    ConvData[1].TrussInfo := TrussInfo;
    RunTrussInfo          := TRUE;
ELSIF ConvData[1].State = E_Outfeed_Conveyor_State.BUILD_IN_PROGRESS THEN
    //bad truss data, index forward or cancel if it's already cleared
    result := RaiseMessageBox(Header   := 'Old truss data detected',
                              Message1 := 'Conveyor has data from previous truss',
                              Message2 := 'Select Clear if conveyor is clear and ready for current truss',
                              Message3 := 'Select Index to send old truss out down the line',
                              Message4 := 'WARNING make sure conveyor is clear or has correct truss on it',
                              Message5 := 'If Index is pressed robot will place once truss is clear',
                              Btn1     := 'Clear',
                              Btn3     := 'Index');

    IF result = 1 THEN
        ConvData[1].State := E_Outfeed_Conveyor_State.IDLE;
    ELSIF result = 3 THEN
        ConvData[1].State := E_Outfeed_Conveyor_State.INDEX_PREP;
    END_IF

END_IF
END_METHOD

(*! @summary This method contains code which will execute when this PackML module is in the <b>Aborted</b> state*)
METHOD PROTECTED Aborted
ControlPendant.Light.Flash();
LightStack.WhiteLight.Flash();
LightStack.Siren.TurnOff();

IF _OutfeedAutostopOK AND _MainSafetyOK THEN
    ChangeState(E_PMLCommand.ePMLCommand_Clear);
END_IF

AllStopped := FALSE;
END_METHOD

METHOD PROTECTED Execute
VAR_INPUT
END_VAR

VAR_INST
    ErrorPresent : BOOL;
	Manual_R_TRIG : R_TRIG;
END_VAR

VAR CONSTANT
	TestConveyorSpeed : UDINT := 500;
END_VAR
ErrorPresent := FALSE;

AllStopped := TRUE;

FOR i := 1 TO _MaxConveyorCount DO
    AllStopped := AllStopped AND (ConvData[i].State = E_Outfeed_Conveyor_State.IDLE OR ConvData[i].State = E_Outfeed_Conveyor_State.OCCUPIED);
END_FOR

IF EnableManualConveyorControl AND AllStopped THEN
    ManualModeActive := TRUE;
    HMIControl();
ELSE
    ManualModeActive := FALSE;

    FOR i := 2 TO _MaxConveyorCount DO
        ErrorPresent := Convey_Motors[i].Error;

        IF ErrorPresent THEN
            EXIT;
        END_IF
    END_FOR

    IF _OutfeedAutostopOK AND _MainSafetyOK AND ErrorPresent = FALSE THEN
        OutfeedConveyorLogic();
    ELSE
        ChangeState(E_PMLCommand.ePMLCommand_Suspend);
    END_IF

    StartUp := FALSE;
    SUPER^.Execute();
END_IF

Manual_R_TRIG(CLK := ManualModeActive);

IF Manual_R_TRIG.Q THEN
    FOR i := 1 TO _MaxConveyorCount DO
        ConvData[i].ManualControlSelected := FALSE;
    END_FOR
END_IF
END_METHOD

METHOD PROTECTED Held
VAR_INPUT
END_VAR
IF _OutfeedAutostopOK AND _MainSafetyOK THEN
    ChangeState(E_PMLCommand.ePMLCommand_Unhold);
END_IF

FOR i := 1 TO _MaxConveyorCount DO
    ConvData[i].SubState := CONV_MOVE_ASSIGN;
END_FOR
END_METHOD

METHOD PROTECTED Idle
VAR_INPUT
END_VAR
IF _OutfeedAutostopOK AND _MainSafetyOK THEN
    ChangeState(E_PMLCommand.ePMLCommand_Start);
END_IF

FOR i := 1 TO _MaxConveyorCount DO
    ConvData[i].SubState := CONV_MOVE_ASSIGN;
END_FOR

EnableManualConveyorControl := FALSE;
END_METHOD

METHOD PROTECTED Stopped
VAR_INPUT
END_VAR
IF _OutfeedAutostopOK AND _MainSafetyOK THEN
    ChangeState(E_PMLCommand.ePMLCommand_Reset);
END_IF

//skip when warm restart detected
RecoveryDetected := NOT StartUp;
END_METHOD

METHOD PROTECTED Suspended
VAR_INPUT
END_VAR
SuspendTON(IN := TRUE, PT := T#2S);

ControlPendant.Light.Flash();
LightStack.WhiteLight.Flash();
LightStack.Siren.TurnOff();

IF _OutfeedAutostopOK AND _MainSafetyOK AND SuspendTON.Q THEN
    ChangeState(E_PMLCommand.ePMLCommand_Unsuspend);
END_IF

FOR i := 1 TO _MaxConveyorCount DO
    ConvData[i].SubState := CONV_MOVE_ASSIGN;
END_FOR

AllStopped := FALSE;
END_METHOD

//! @summary This method monitors <b>components</b> within this PackML module and initiates fault responses as required
METHOD PROTECTED ComponentMonitor : BOOL
VAR
    AlarmResponses : ARRAY[0..4] OF E_AlarmResponse; //Temporary response array
    i              : UDINT;
END_VAR

//! @description This method is called cyclically by <c>CyclicLogic()</c>
FOR i := 2 TO NumberOfComponents DO
    IF _CurrentState <> E_PMLState.ePMLState_Aborted AND
       _CurrentState <> E_PMLState.ePMLState_Aborting AND
       _CurrentState <> E_PMLState.ePMLState_Clearing AND
       _CurrentState <> E_PMLState.ePMLState_Suspended AND
       _CurrentState <> E_PMLState.ePMLState_Unsuspending AND
       _CurrentState <> E_PMLState.ePMLState_Held AND
       _CurrentState <> E_PMLState.ePMLState_Unholding AND
       _CurrentState <> E_PMLState.ePMLState_Stopped AND
       _CurrentState <> E_PMLState.ePMLState_Stopping THEN
        AlarmResponses := ipComponents[i].ParentResponseDefinitions;

        CASE AlarmResponses[ipComponents[i].CurrentAlarmSeverity] OF
            E_AlarmResponse.Abort_ImmediateError:
                SuspendImmediate();

            E_AlarmResponse.Abort_Immediate:
                SuspendControlled();

            E_AlarmResponse.Stop_Immediate:
                StopImmediate();

            E_AlarmResponse.Stop_Controlled:
                StopControlled();

            E_AlarmResponse.Hold_Immediate:
                HoldImmediate();

            E_AlarmResponse.Hold_Controlled:
                HoldControlled();

            E_AlarmResponse.Suspend_Immediate:
                SuspendImmediate();

            E_AlarmResponse.Suspend_Controlled:
                SuspendControlled();

            E_AlarmResponse.NoResponse:
                ;
        END_CASE
    ELSIF _CurrentState = E_PMLState.ePMLState_Stopped OR _CurrentState = E_PMLState.ePMLState_Stopping THEN
        AlarmResponses := ipComponents[i].ParentResponseDefinitions;

        CASE AlarmResponses[ipComponents[i].CurrentAlarmSeverity] OF
            E_AlarmResponse.Abort_ImmediateError:
                AbortImmediateError(ipComponents[i].Name, FALSE);

            E_AlarmResponse.Abort_Immediate:
                AbortImmediate();

            E_AlarmResponse.NoResponse:
                ;
        END_CASE
    END_IF
END_FOR
END_METHOD

METHOD PROTECTED CreateEvents
VAR_INPUT
END_VAR
F_CreateAllEventsInClass(Alarms     := OutfeedJigAlarms,
                         ClassSize  := SIZEOF(TC_EVENTS.Outfeed_Jig),
                         pInitEvent := ADR(TC_EVENTS.Outfeed_Jig.InitReferenceEvent),
                         Prefix     := _Name);

SUPER^.CreateEvents();
END_METHOD

METHOD HMIControl
VAR_INPUT
END_VAR

VAR
	AllReset : BOOL;
END_VAR
IF ManualReset = FALSE THEN

    FOR i := 1 TO _MaxConveyorCount DO

        IF ManualControlConveyFWD THEN
            IF ConvData[i].ManualControlSelected AND ConvData[i].State = E_Outfeed_Conveyor_State.IDLE THEN
                Convey_Motors[i].MoveVelocity(ManualConveyorSpeed, TRUE);
            ELSE
                IF Convey_Motors[i].Busy THEN
                    Convey_Motors[i].Stop();
                END_IF
            END_IF
        ELSIF ManualControlConveyREV THEN
            IF ConvData[i].ManualControlSelected AND ConvData[i].State = E_Outfeed_Conveyor_State.IDLE THEN
                Convey_Motors[i].MoveVelocity(-ManualConveyorSpeed, TRUE);
            ELSE
                IF Convey_Motors[i].Busy THEN
                    Convey_Motors[i].Stop();
                END_IF
            END_IF
        ELSE

            IF Convey_Motors[i].Busy THEN
                Convey_Motors[i].Stop();
            END_IF
        END_IF

    END_FOR
ELSE
	AllReset := TRUE;
    FOR i := 1 TO _MaxConveyorCount DO
       AllReset := MotorResetAndEnable(Convey_Motors[i]) AND AllReset; 
    END_FOR
	IF AllReset THEN
		ManualReset := FALSE;
	END_IF
END_IF
END_METHOD

METHOD IndexFull : BOOL
VAR_INPUT
END_VAR

VAR_INST
    SubState : USINT := 0;
END_VAR
IndexFull := FALSE;

CASE SubState OF
    0:
        IF ConvData[1].State = E_Outfeed_Conveyor_State.BUILD_IN_PROGRESS THEN
            ConvData[1].State := E_Outfeed_Conveyor_State.INDEX_PREP;
            SubState          := 10;
        END_IF

    10:
        IndexFull := TRUE;
        SubState  := 0;

END_CASE
END_METHOD

METHOD IndexHalf : BOOL
VAR_INPUT
END_VAR

VAR_INST
    SubState : USINT := 0;
END_VAR
IndexHalf := FALSE;

CASE SubState OF
    0:
        IF ConvData[1].State = E_Outfeed_Conveyor_State.BUILD_IN_PROGRESS THEN
            ConvData[1].State := E_Outfeed_Conveyor_State.INDEX_HALF_PREP;
        ELSE
            //waiting for conveyor 1 to be in a good spot
        END_IF

        IF ConvData[1].State = E_Outfeed_Conveyor_State.INDEXING_HALF THEN
            SubState := 10;
        END_IF

    10:
        IF ConvData[1].State = E_Outfeed_Conveyor_State.BUILD_IN_PROGRESS THEN
            IndexHalf := TRUE;
            SubState  := 0;
        END_IF

END_CASE
END_METHOD

//! @summary Basic module initialization logic
METHOD PROTECTED Initialize : BOOL;
VAR
    i                        : UDINT;
    varInfo                  : __SYSTEM.VAR_INFO;
    AllSubUnitsInitialized   : BOOL := TRUE;
    AllComponentsInitialized : BOOL := TRUE;
    emptyTrussInfo           : ST_TrussInfo;

END_VAR

//! @description This method is called by <c>CyclicLogic()</c> as required
CASE DescendantSequenceState OF
    0:
        RegisterComponent(Shift_Motors);
        RegisterComponent(ControlPendant);
        RegisterComponent(LightStack);

        FOR i := 1 TO _MaxConveyorCount DO
            RegisterComponent(Convey_Motors[i]);
            //RegisterComponent(Convey_Sensors[i]);
            ConvData[i].SubState           := E_Outfeed_Conveyor_SubState.CONV_MOVE_ASSIGN;
            ConvData[i].HalfIndexCompleted := FALSE;
            ConvData[i].ReadyForSlideOut   := FALSE;
            ConvData[i].ReadyToIndex       := FALSE;
            ConvData[i].ReadyToIndexHalf   := FALSE;
            ConvData[i].ReadyToOutfeed     := FALSE;
            ConvData[i].ReadyToReceive     := FALSE;
        END_FOR

        LogModeChanges  := FALSE;
        LogStateChanges := FALSE;

        RegisterExternalController(Controller := fbControlSourceHMI);
        fbControlSourceHMI.CyclicLogic();

        //Copy Mode names

        FOR i := 1 TO 3 DO
            ModeNames[i] := F_UnitModeToString(UDINT_TO_DINT(i));
        END_FOR

        DescendantSequenceState := 1;

    1:
        CreateEvents();

        IF SUPER^.Initialize() THEN
            DescendantSequenceState := 2;
        END_IF

    2:
        Initialize := TRUE;

END_CASE
END_METHOD

METHOD PROTECTED Monitoring
VAR_INPUT
END_VAR
///////////////////////////////////////////////////////////////////////////////
// 5. Outfeed autostop dropped
///////////////////////////////////////////////////////////////////////////////
IF (NOT OutfeedJigAlarms[E_Outfeed_Jig.OutfeedSafetyDropped].bRaised) AND NOT _OutfeedAutostopOK THEN
    // Raise alarm if Infeed is taking a long time to get a board
    OutfeedJigAlarms[E_Outfeed_Jig.OutfeedSafetyDropped].Raise(0);
ELSIF OutfeedJigAlarms[E_Outfeed_Jig.OutfeedSafetyDropped].bRaised AND _OutfeedAutostopOK THEN
    // Clear when a board is found
    OutfeedJigAlarms[E_Outfeed_Jig.OutfeedSafetyDropped].Clear(0, 0);
END_IF;

///////////////////////////////////////////////////////////////////////////////
// 5. Outfeed autostop dropped
///////////////////////////////////////////////////////////////////////////////
IF (NOT OutfeedJigAlarms[E_Outfeed_Jig.IndexingBlocked].bRaised) AND IndexingBlockedAlarm THEN
    // Raise alarm if Infeed is taking a long time to get a board
    OutfeedJigAlarms[E_Outfeed_Jig.IndexingBlocked].Raise(0);
ELSIF OutfeedJigAlarms[E_Outfeed_Jig.IndexingBlocked].bRaised AND NOT IndexingBlockedAlarm THEN
    // Clear when a board is found
    OutfeedJigAlarms[E_Outfeed_Jig.IndexingBlocked].Clear(0, 0);
END_IF;

//////////////////////////////////////////////////////////////////////////
// Wrap-up: Evaluate overall severity, then run the extended Monitoring
//////////////////////////////////////////////////////////////////////////
_CurrentAlarmSeverity := TcEventSeverity.Verbose;
_CurrentAlarmSeverity := F_GetMaxSeverityRaised(Alarms := OutfeedJigAlarms, CurrentSeverity := _CurrentAlarmSeverity);

// Finally, run the extended monitoring
// SUPER^.Monitoring();
END_METHOD

METHOD MotorsInit : BOOL
VAR_INPUT
END_VAR
MotorsInit := TRUE;

FOR i := 1 TO _MaxConveyorCount DO
    IF (_MainSafetyOK AND _AutostopOK AND i = 1) OR i > 1 THEN
        MotorsInit := MotorResetAndEnable(Convey_Motors[i]) AND MotorsInit AND Shift_Motors.Reset();
    END_IF
END_FOR
END_METHOD

METHOD NewTrussInfo : BOOL
VAR_INPUT
    ConveyorIndex : USINT;
    NewTrussData  : ST_TrussInfo;
END_VAR

VAR
    i              : USINT;
    EmptyBoardData : ST_PickPlace;
    EmptyTrussInfo : ST_TrussInfo;
END_VAR
FOR i := 1 TO 50 DO
    IF ConvData[1].BoardsPresent[i].ID = '' AND ConvData[1].BoardsPresent[i].Length = 0 THEN
        ConvData[1].BoardsPresent[i] := EmptyBoardData;
    END_IF
END_FOR

ConvData[1].TrussInfo := NewTrussData;
END_METHOD

METHOD OutfeedConveyorLogic : BOOL
VAR_INPUT
END_VAR

VAR
    EmptyBoardsPresent : ARRAY[1..50] OF ST_PickPlace;
    EmptyTrussInfo     : ST_TrussInfo;
    TempString         : STRING;
END_VAR

VAR_INST
    Previous_SubState : ARRAY[1..7] OF E_Outfeed_Conveyor_SubState;
    ClearConveyorTON  : TON;
    Previous_State    : ARRAY[1..7] OF E_Outfeed_Conveyor_State;
    Alarm_TON         : ARRAY[1..7] OF TON;
END_VAR
LightStack.WhiteLight.TurnOn();
ControlPendant.Light.TurnOff();

FOR i := 1 TO _MaxConveyorCount DO
    CASE ConvData[i].State OF
        E_Outfeed_Conveyor_State.IDLE:
            ConvData[i].SubState := CONV_MOVE_ASSIGN;

            // check to see if index is requested
            Alarm_TON[i](IN := FALSE, PT := T#5S);

            IF i = _MaxConveyorCount THEN
                ClearConveyorTON(IN := FALSE, PT := T#1000MS);
                LightStack.Siren.TurnOff();
                LightStack.AmberLight.TurnOff();
            END_IF

            IF i > 1 THEN
                IF ConvData[i - 1].ReadyToIndex THEN
                    ConvData[i].State := E_Outfeed_Conveyor_State.RECEIVE_PREP;
                END_IF
            END_IF

        E_Outfeed_Conveyor_State.RECEIVE_PREP:
            // assign absolute position based off relative distance, also sync up with indexing conveyor

            IF Convey_Motors[i].Enabled AND Convey_Motors[i].Error = FALSE THEN
                ConvData[i].TargetPos          := Convey_Motors[i].ActualPosition + ConvData[i].ConveyorLength;
                ConvData[i - 1].ReadyToReceive := TRUE;

                IF i = _MaxConveyorCount AND Shift_Motors.Retracted THEN
                    ConvData[i].State := E_Outfeed_Conveyor_State.RECEIVING;
                ELSE
                    ConvData[i].State := E_Outfeed_Conveyor_State.RECEIVING;
                END_IF
            ELSE
                MotorResetAndEnable(Convey_Motors[i]);
            END_IF

        E_Outfeed_Conveyor_State.RECEIVING:

            // execute movement to position go to RESET when done

            CASE ConvData[i].SubState OF
                CONV_MOVE_ASSIGN:
                    IF i = 2 THEN
                        IF _AutostopOK AND Convey_Motors[i - 1].Axis.Status.DiscreteMotion THEN
                            Convey_Motors[i].MoveAbsolute(ConvData[i].TargetPos, TRUE);
                            ConvData[i].SubState := CONV_MOVE_DONE_CHECK;
                        END_IF
                    ELSE
                        Convey_Motors[i].MoveAbsolute(ConvData[i].TargetPos, TRUE);
                        ConvData[i].SubState := CONV_MOVE_DONE_CHECK;
                    END_IF

                CONV_MOVE_DONE_CHECK:
                    IF Convey_Motors[i].InPosition AND NOT Convey_Motors[i].Busy THEN
                        ConvData[i].SubState := CONV_DATA_CONFIRMATION;
                    ELSIF Convey_Motors[i].Error OR (i = 2 AND (_AutostopOK = FALSE)) THEN
                        ConvData[i].SubState := CONV_RESET_MOTOR;
                    END_IF

                CONV_DATA_CONFIRMATION:
                    Alarm_TON[i](IN := TRUE, PT := T#5S);

                    IF ConvData[i].TrussInfo.TrussID <> '' THEN
                        ConvData[i].SubState := CONV_MOVE_ASSIGN;
                        ConvData[i].State    := E_Outfeed_Conveyor_State.OCCUPIED;
                        Alarm_TON[i](IN := FALSE, PT := T#5S);
                    END_IF

                    Convey_Motors[i].AlarmRaiseBasic(alarm := E_OutfeedConveyor.NoTrussData, raise := Alarm_TON[i].Q);

                CONV_RESET_MOTOR:
                    IF MotorResetAndEnable(Convey_Motors[i]) THEN
                        ConvData[i].SubState := CONV_MOVE_ASSIGN;
                    END_IF
            END_CASE

        E_Outfeed_Conveyor_State.OCCUPIED:
            // check to see if boards can be moved forward

            IF i < _MaxConveyorCount THEN
                IF ConvData[i + 1].State = E_Outfeed_Conveyor_State.IDLE THEN
                    ConvData[i].State := E_Outfeed_Conveyor_State.INDEX_PREP;
                END_IF
            ELSE
                //turn on lights and permissions for extending and retracting conveyor out over table button pressed to clear data and let them retract

                ControlPendant.Light.TurnOn();
                LightStack.AmberLight.TurnOn();
                Shift_Motors.Jog(JogFW := ControlPendant.ExtendSlideout.Button_Pressed, JogBW := ControlPendant.RetractSlideout.Button_Pressed);

                IF Shift_Motors.Retracted = FALSE THEN
                    ConvData[i].State := E_Outfeed_Conveyor_State.RESET;
                ELSIF _InSimulation THEN
                    ConvData[i].State := E_Outfeed_Conveyor_State.AUTO_RETRACT;
                END_IF
            END_IF

        E_Outfeed_Conveyor_State.INDEX_HALF_PREP:
            ConvData[i].TargetPos := Convey_Motors[i].ActualPosition + (ConvData[i].ConveyorLength / 2);
            Alarm_TON[i](IN := TRUE, PT := T#5S);

            // assign absolute position based off relative distance, also sync up with receiving conveyor
            IF Convey_Motors[i].Enabled AND Convey_Motors[i].Error = FALSE THEN
                ConvData[i].State := E_Outfeed_Conveyor_State.INDEXING_HALF;
                Alarm_TON[i](IN := FALSE, PT := T#5S);
            ELSE
                IF _MainSafetyOK AND ((i > 1 AND _OutfeedAutostopOK) OR (i = 1 AND _AutostopOK)) THEN
                    MotorResetAndEnable(Convey_Motors[i]);
                END_IF
            END_IF

            IndexingBlockedAlarm := Alarm_TON[i].Q;

        E_Outfeed_Conveyor_State.INDEXING_HALF:
            // execute movement to position go to RESET when done

            CASE ConvData[i].SubState OF
                CONV_MOVE_ASSIGN:
                    Convey_Motors[i].MoveAbsolute(ConvData[i].TargetPos, TRUE);
                    ConvData[i].SubState := CONV_MOVE_DONE_CHECK;

                CONV_MOVE_DONE_CHECK:
                    IF Convey_Motors[i].InPosition AND NOT Convey_Motors[i].Busy THEN
                        ConvData[i].State    := E_Outfeed_Conveyor_State.BUILD_IN_PROGRESS;
                        ConvData[i].SubState := CONV_MOVE_ASSIGN;
                    ELSIF Convey_Motors[i].Error THEN
                        ConvData[i].SubState := CONV_RESET_MOTOR;
                    END_IF

                CONV_RESET_MOTOR:
                    IF MotorResetAndEnable(Convey_Motors[i]) THEN
                        ConvData[i].SubState := CONV_MOVE_ASSIGN;
                    END_IF

            END_CASE

        E_Outfeed_Conveyor_State.INDEX_PREP:
            Alarm_TON[i](IN := TRUE, PT := T#5S);

            IndexingBlockedAlarm := Alarm_TON[i].Q;

            IF Convey_Motors[i].Enabled AND Convey_Motors[i].Error = FALSE THEN
                ConvData[i].TargetPos    := Convey_Motors[i].ActualPosition + ConvData[i].ConveyorLength;
                ConvData[i].ReadyToIndex := TRUE;

                // assign absolute position based off relative distance, also sync up with receiving conveyor
                IF ConvData[i + 1].State = E_Outfeed_Conveyor_State.RECEIVING THEN
                    IF Convey_Motors[i].Enabled AND Convey_Motors[i].Error = FALSE THEN
                        ConvData[i].State := E_Outfeed_Conveyor_State.INDEXING;
                        Alarm_TON[i](IN := FALSE, PT := T#5S);
                    ELSE
                        MotorResetAndEnable(Convey_Motors[i]);
                    END_IF
                END_IF
            ELSE
                IF _MainSafetyOK AND ((i > 1 AND _OutfeedAutostopOK) OR (i = 1 AND _AutostopOK)) THEN
                    MotorResetAndEnable(Convey_Motors[i]);
                END_IF
            END_IF

        E_Outfeed_Conveyor_State.INDEXING:
            // execute movement to position go to RESET when done

            CASE ConvData[i].SubState OF
                CONV_MOVE_ASSIGN:
                    IF i = 1 THEN
                        IF _AutostopOK THEN
                            Convey_Motors[i].MoveAbsolute(ConvData[i].TargetPos, TRUE);
                            ConvData[i].SubState := CONV_MOVE_DONE_CHECK;
                        END_IF
                    ELSE
                        Convey_Motors[i].MoveAbsolute(ConvData[i].TargetPos, TRUE);
                        ConvData[i].SubState := CONV_MOVE_DONE_CHECK;
                    END_IF

                CONV_MOVE_DONE_CHECK:
                    IF Convey_Motors[i].InPosition AND NOT Convey_Motors[i].Busy THEN
                        ConvData[i].SubState := CONV_DATA_CONFIRMATION;
                    ELSIF Convey_Motors[i].Error OR (i = 1 AND _AutostopOK = FALSE) THEN
                        ConvData[i].SubState := CONV_RESET_MOTOR;
                    END_IF

                CONV_DATA_CONFIRMATION:
                    ConvData[i + 1].BoardsPresent := ConvData[i].BoardsPresent;
                    ConvData[i + 1].TrussInfo     := ConvData[i].TrussInfo;

                    IF ConvData[i + 1].State = E_Outfeed_Conveyor_State.OCCUPIED THEN
                        ConvData[i].State    := E_Outfeed_Conveyor_State.RESET;
                        ConvData[i].SubState := CONV_MOVE_ASSIGN;

                        ConvData[i].ReadyToIndex := FALSE;
                    END_IF

                CONV_RESET_MOTOR:
                    IF MotorResetAndEnable(Convey_Motors[i]) THEN
                        ConvData[i].SubState := CONV_MOVE_ASSIGN;
                    END_IF
            END_CASE

        E_Outfeed_Conveyor_State.RESET:
            // reset data and start at IDLE
            ConvData[i].SubState := CONV_MOVE_ASSIGN;

            IF i < _MaxConveyorCount THEN
                IF Convey_Motors[i].SimHoming(Motor := Convey_Motors[i], SimPos := 0) THEN
                    ConvData[i].BoardsPresent := EmptyBoardsPresent;
                    ConvData[i].TrussInfo     := EmptyTrussInfo;
                    ConvData[i].ReadyToIndex  := FALSE;

                    ConvData[i].State := E_Outfeed_Conveyor_State.IDLE;
                END_IF
            ELSE
                //turn on lights and permissions for extending conveyor out over table, clear data and let them retract

                ClearConveyorTON(IN := ControlPendant.ClearConveyor.Button_Pressed AND ControlPendant.RetractSlideout.Button_Pressed, PT := T#250MS);

                ControlPendant.Light.TurnOn();
                LightStack.AmberLight.TurnOn();
                Shift_Motors.Jog(JogFW := ControlPendant.ExtendSlideout.Button_Pressed, JogBW := ControlPendant.RetractSlideout.Button_Pressed);

                IF ClearConveyorTON.Q THEN
                    ConvData[i].State := E_Outfeed_Conveyor_State.AUTO_RETRACT;
                END_IF

            END_IF

        E_Outfeed_Conveyor_State.AUTO_RETRACT:
            LightStack.AmberLight.Flash();
            LightStack.Siren.Flash();

            IF Shift_Motors.Retracted = FALSE AND _InSimulation = FALSE THEN
                Shift_Motors.Jog(JogFW := FALSE, JogBW := TRUE);

                IF ControlPendant.ExtendSlideout.Button_Pressed THEN
                    ConvData[i].State := E_Outfeed_Conveyor_State.RESET;
                END_IF
            ELSE
                Shift_Motors.Jog(JogFW := FALSE, JogBW := FALSE);

                IF Convey_Motors[i].SimHoming(Motor := Convey_Motors[i], SimPos := 0) THEN
                    ConvData[i].BoardsPresent := EmptyBoardsPresent;
                    ConvData[i].TrussInfo     := EmptyTrussInfo;
                    ConvData[i].ReadyToIndex  := FALSE;
                    ConvData[i].State         := E_Outfeed_Conveyor_State.IDLE;
                    ControlPendant.Light.TurnOff();
                END_IF
            END_IF

        E_Outfeed_Conveyor_State.ERROR:

        // Conveyor errored out, prevent indexing or receiving from other conveyors
    END_CASE

    IF ConvData[i].State <> Previous_State[i] THEN
        TempString := '';
        TempString := CONCAT(TempString, 'Conveyor ');
        TempString := CONCAT(TempString, UDINT_TO_STRING(i));
        TempString := CONCAT(TempString, ' State change to: ');
        Trace(CONCAT(TempString, TO_STRING(ConvData[i].State)));
    END_IF

    Previous_State[i] := ConvData[i].State;

    IF ConvData[i].SubState <> Previous_SubState[i] THEN
        TempString := '';
        TempString := CONCAT(TempString, 'Conveyor ');
        TempString := CONCAT(TempString, UDINT_TO_STRING(i));
        TempString := CONCAT(TempString, ' SubState change to: ');
        Trace(CONCAT(TempString, TO_STRING(ConvData[i].SubState)));
    END_IF

    Previous_SubState[i] := ConvData[i].SubState;

END_FOR
END_METHOD

METHOD PopulateBoardToArray : BOOL
VAR_INPUT
    ConveyorIndex : USINT;
    NewBoardData  : ST_PickPlace;
END_VAR

VAR
    i : USINT;
END_VAR
FOR i := 1 TO 50 DO
    IF ConvData[1].BoardsPresent[i].ID = '' AND ConvData[1].BoardsPresent[i].Length = 0 THEN
        ConvData[1].BoardsPresent[i] := NewBoardData;
        EXIT;
    END_IF
END_FOR
END_METHOD

PROPERTY AutostopOK : bool
SET
_AutostopOK := AutostopOK;
END_SET
END_PROPERTY

PROPERTY MainSafetyOK : bool
SET
_MainSafetyOK := MainSafetyOK;
END_SET
END_PROPERTY

PROPERTY MaxConveyorCount : USINT
SET
_MaxConveyorCount := MaxConveyorCount;
END_SET
END_PROPERTY

PROPERTY OutfeedAutostopOK : bool
SET
_OutfeedAutostopOK := OutfeedAutostopOK;
END_SET
END_PROPERTY

PROPERTY OutfeedConveyorStatus : ST_OutfeedConveyorStatus
GET
OutfeedConveyorStatus := _OutfeedConveyorStatus;
END_GET
END_PROPERTY

PROPERTY ParentState : E_PMLState
SET
_ParentState := ParentState;
END_SET
END_PROPERTY

PROPERTY PickPlace_Done_ENUM : E_WaitSync
SET
_PickPlace_Done_ENUM := PickPlace_Done_ENUM;
END_SET
END_PROPERTY

PROPERTY PickPlace_Ready_ENUM : E_WaitSync
SET
_PickPlace_Ready_ENUM := PickPlace_Ready_ENUM;
END_SET
END_PROPERTY

END_FUNCTION_BLOCK

// Machine/EquipmentModules/Functional Layer/FB_Preplate
FUNCTION_BLOCK FB_Preplate EXTENDS FB_EquipmentModule_SR
VAR
    // Sub module definitions here

    // List of sub modules

    // Component definitions here
    Racks       : ARRAY[1..NUM_OF_PREPLATE_RACKS] OF FB_Component_Preplate_Rack;
    ManDoorLock : FB_Component_Indicator;

END_VAR

VAR CONSTANT

    // Report parameters 

    //Alarms
    NUM_OF_PREPLATE_RACKS : UDINT := 5;

    PREPLATE_ALARM_COUNT : INT := 6;
END_VAR

VAR CONSTANT

    SS_OPEN_DOORS  : INT := 200;
    SS_CLOSE_DOORS : INT := 201;
END_VAR

METHOD CyclicLogic
VAR_INPUT
END_VAR

VAR
    LowLimit  : STRING;
    HighLimit : STRING;
END_VAR
IF NOT _InitComplete THEN
    _InitComplete := Initialize();
    RETURN;
END_IF

SUPER^.CyclicLogic();

IF _CurrentState = E_PMLState.ePMLState_Execute OR
   _CurrentState = E_PMLState.ePMLState_Unholding OR
   _CurrentState = E_PMLState.ePMLState_Unsuspending THEN

    ManDoorLock.TurnOn();
ELSE
    ManDoorLock.TurnOff();
END_IF

IF _CurrentState <> E_PMLState.ePMLState_Execute THEN
    FOR i := 1 TO NUM_OF_PREPLATE_RACKS DO
        Racks[i].Executing := FALSE;
    END_FOR
END_IF

Racks[1].LinkBlocked := Racks[2].Blocked;
Racks[2].LinkBlocked := Racks[1].Blocked;
Racks[3].LinkBlocked := Racks[4].Blocked;
Racks[4].LinkBlocked := Racks[3].Blocked OR Racks[4].Blocked;
Racks[5].LinkBlocked := Racks[4].Blocked;
;
IF NOT Racks[1].IsAvailable() THEN
	Racks[2].Disable();
END_IF

IF NOT Racks[2].IsAvailable() THEN
	Racks[1].Disable();
END_IF

IF NOT Racks[3].IsAvailable() THEN
	Racks[4].Disable();
END_IF

IF NOT Racks[4].IsAvailable() THEN
	Racks[3].Disable();
END_IF

CyclicLogicSimulation();
END_METHOD

(*! @summary This method contains code which will execute when this PackML module is in the <b>Execute</b> state*)
METHOD PROTECTED Execute
ManDoorLock.TurnOn();

FOR i := 1 TO NUM_OF_PREPLATE_RACKS DO
    Racks[i].Executing := TRUE;
END_FOR
END_METHOD

METHOD HMIControl
VAR_INPUT
END_VAR
END_METHOD

//! @summary Basic module initialization logic
METHOD PROTECTED Initialize : BOOL;
VAR
    i                        : UDINT;
    varInfo                  : __SYSTEM.VAR_INFO;
    AllSubUnitsInitialized   : BOOL := TRUE;
    AllComponentsInitialized : BOOL := TRUE;
END_VAR

//! @description This method is called by <c>CyclicLogic()</c> as required
Initialize := FALSE;

CASE DescendantSequenceState OF
    0:
        FOR i := 1 TO NUM_OF_PREPLATE_RACKS DO
            RegisterComponent(Racks[i]);
        END_FOR

        _LogModeChanges         := FALSE;
        _LogStateChanges        := FALSE;
        DescendantSequenceState := DescendantSequenceState + 10;

    10:
        //Setup Custom modes here

        (*CustomModes(eMode                          :=,
                    sName                          :=,
                    bDisableClearing               :=,
                    bDisableStarting               :=,
                    bDisableSuspended              :=,
                    bDisableStopping               :=,
                    bDisableAborting               :=,
                    bDisableHolding                :=,
                    bDisableHeld                   :=,
                    bDisableUnholding              :=,
                    bDisableSuspending             :=,
                    bDisableUnsuspending           :=,
                    bDisableResetting              :=,
                    bDisableIdle                   :=,
                    bDisableCompleting             :=,
                    bDisableComplete               :=,
                    bEnableUnitModeChangeStopped   :=,
                    bEnableUnitModeChangeIdle      :=,
                    bEnableUnitModeChangeSuspended :=,
                    bEnableUnitModeChangeExecute   :=,
                    bEnableUnitModeChangeAborted   :=,
                    bEnableUnitModeChangeHeld      :=,
                    bEnableUnitModeChangeComplete  :=,
                    bError                         =>,
                    nErrorId                       =>);*)

        DescendantSequenceState := DescendantSequenceState + 10;

    20:
        //Copy Mode names

        FOR i := 1 TO 3 DO
            ModeNames[i] := F_UnitModeToString(UDINT_TO_DINT(i));
        END_FOR

        RegisterExternalController(Controller := fbControlSourceHMI);
        fbControlSourceHMI.CyclicLogic();
        DescendantSequenceState := DescendantSequenceState + 10;

    30:
        //Call the Super

        IF SUPER^.Initialize() THEN
            DescendantSequenceState := DescendantSequenceState + 10;
        END_IF

    40:
        Initialize := TRUE;
END_CASE
END_METHOD

PROPERTY PUBLIC InAuto : BOOL
GET
END_GET
SET
FOR i := 1 TO NUM_OF_PREPLATE_RACKS DO
    Racks[i].InAuto := InAuto;
END_FOR
END_SET
END_PROPERTY

END_FUNCTION_BLOCK

// Machine/EquipmentModules/Functional Layer/FB_Press
FUNCTION_BLOCK FB_Press EXTENDS FB_EquipmentModule_SR
VAR
    // Sub module definitions here

    // List of sub modules

    ipSubModules_Init : ARRAY[1..Parameters_PackML_Base.MAX_NO_OF_SUBMODULES] OF I_PackML_BaseModule := [];

    // Component definitions here

    Top_Press    : FB_Component_BasicSlaveAxis_SoE := (Name := 'Top Press');
    Bottom_Press : FB_Component_BasicSlaveAxis_SoE := (Name := 'Bottom Press');

    Top_PressCmds_Extra    : ST_MotorControls_NonStandard;
    Bottom_PressCmds_Extra : ST_MotorControls_NonStandard;

    //Data for recipe

    TopPressRecipe    : ST_PressRecipe;
    BottomPressRecipe : ST_PressRecipe;
    Plates            : ST_Plates;
    DetailIndex       : UDINT := 1;
    Detail_Step       : E_Press_States;

    _NailplateCountData_Ready : BOOL;
    _NailplateCountData_Sent  : BOOL;
    _DriveMode                : SPT_Motion_Control.E_DriveOperationMode;
    _DoublePickDataToPass     : BOOL;
    _DoublePickData_Ready     : BOOL;
    _DoublePickData_Sent      : BOOL;
    _BoardDataToPass          : ST_BoardInfo;
END_VAR

VAR CONSTANT

    // Report parameters 

    FAULTID  : INT := 1; //Fault number 
    CURRTEMP : INT := 2; // current temperature of the sealing bar 
    CURRPOS  : INT := 3; // current position of the sealing bar  

    //Alarms

    PREPLATE_ALARM_COUNT : INT := 6;
END_VAR

VAR
    FB_Reset_SoE_Drive : FB_SoEReset;

    //Robot Signals

    RobotClearOfPress AT %I* : BOOL := TRUE;

    _NailplateDataToPass : ST_PlateInfo;

    TopPressDriveOpMode_Read    : SPT_Motion_Control.MC_ReadDriveOperationMode;
    TopPressDriveOpMode_Write   : SPT_Motion_Control.MC_WriteDriveOperationMode;
    TopPressDriveOpMode_Options : SPT_Motion_Control.ST_DriveOperationModeOptions;

    BottomPressDriveOpMode_Read    : SPT_Motion_Control.MC_ReadDriveOperationMode;
    BottomPressDriveOpMode_Write   : SPT_Motion_Control.MC_WriteDriveOperationMode;
    BottomPressDriveOpMode_Options : SPT_Motion_Control.ST_DriveOperationModeOptions;

    _PressRobotPermissionToEnter : ST_MediatorInterface;
END_VAR

METHOD CyclicLogic
VAR_INPUT
END_VAR

VAR
    LowLimit  : STRING;
    HighLimit : STRING;
END_VAR
IF NOT _InitComplete THEN
    _InitComplete := Initialize();
    RETURN;
END_IF

AllowHMIControl(ThisModuleOnly:=FALSE);

SUPER^.CyclicLogic();
CyclicLogicSimulation();

BottomPressRecipe.AtTop := Bottom_Press.ActualPosition < BottomPressRecipe.OpenPosition + 10;
TopPressRecipe.AtTop    := Top_Press.ActualPosition < TopPressRecipe.OpenPosition + 10;

BottomPressRecipe.AtWork := Bottom_Press.ActualPosition > BottomPressRecipe.ClosedPosition - 10;
TopPressRecipe.AtWork    := Top_Press.ActualPosition > TopPressRecipe.ClosedPosition - 10;

BottomPressRecipe.State_Str := TO_STRING(BottomPressRecipe.State);
BottomPressRecipe.State_Previous_Str := TO_STRING(BottomPressRecipe.State_Previous);
BottomPressRecipe.State_Response_Str := TO_STRING(BottomPressRecipe.State_Response);

TopPressRecipe.State_Str := TO_STRING(TopPressRecipe.State);
TopPressRecipe.State_Previous_Str := TO_STRING(TopPressRecipe.State_Previous);
TopPressRecipe.State_Response_Str := TO_STRING(TopPressRecipe.State_Response);
END_METHOD

METHOD PROTECTED Aborting
VAR_INPUT
END_VAR
// CASE SequenceState OF
//     0:
//         NoStateTasksToComplete := FALSE;
// 
//         IF Bottom_Press.Enabled AND NOT Bottom_Press.Error AND Top_Press.Enabled AND NOT Top_Press.Error THEN
//             SequenceState := SequenceState + 10;
//             Trace('SequenceState: 10 - Both presses enabled'); // Log state transition when both presses are enabled
//         ELSE
//             SequenceState := 50;
//             Trace('SequenceState: 50 - One or both presses not enabled'); // Log state transition when one or both presses are not enabled
//         END_IF
// 
//     10:
//         Bottom_Press.Velocity     := BottomPressRecipe.Axis.Velocity;
//         Bottom_Press.Acceleration := BottomPressRecipe.Axis.Acceleration;
//         Bottom_Press.MoveAbsolute(Position := BottomPressRecipe.OpenPosition, TRUE);
//         SequenceState := SequenceState + 10;
//         Trace('SequenceState: 20 - Main press moving to open position'); // Log state transition and main press movement
//     20:
//         IF Bottom_Press.InPosition AND NOT Bottom_Press.Busy THEN
//             SequenceState := SequenceState + 10;
//             Trace('SequenceState: 30 - Main press in position'); // Log state transition when main press is in position
//         END_IF
// 
//     30:
//         Top_Press.Velocity     := TopPressRecipe.Axis.Velocity;
//         Top_Press.Acceleration := TopPressRecipe.Axis.Acceleration;
//         Top_Press.MoveAbsolute(Position := TopPressRecipe.OpenPosition, TRUE);
//         SequenceState := SequenceState + 10;
//         Trace('SequenceState: 40 - Aux press moving to open position'); // Log state transition and aux press movement
//     40:
//         IF Top_Press.InPosition AND NOT Top_Press.Busy THEN
//             SequenceState := SequenceState + 10;
//             Trace('SequenceState: 50 - Aux press in position'); // Log state transition when aux press is in position
//         END_IF
// 
//     50:
//         IF Bottom_Press.Error THEN
//             Bottom_Press.Reset();
//         END_IF
// 
//         IF Top_Press.Error THEN
//             Top_Press.Reset();
//         END_IF
// 
//         Bottom_Press.Stop();
//         Top_Press.Stop();
// 
//         IF Bottom_Press.Stopped AND Top_Press.Stopped THEN
//             SequenceState := SequenceState + 10;
//             Trace('SequenceState: 60 - Both presses stopped'); // Log state transition when both presses are stopped
//         END_IF
// 
//     60:
//         // Disable here
//         Bottom_Press.Disable();
//         Top_Press.Disable();
//         //Trace('SequenceState: 60 - Both presses disabled'); // Log presses disabled state
// 
//         // Check not enabled here
//         IF (NOT Bottom_Press.Enabled) AND (NOT Top_Press.Enabled) THEN
//             SequenceState := SequenceState + 10;
//             Trace('SequenceState: 70 - Both presses not enabled'); // Log state transition when both presses are not enabled
//         END_IF
// 
//     70:
//         StateTasksComplete := TRUE;
// 
//     //Trace('StateTasksComplete: TRUE'); // Log state tasks completion
// END_CASE

Bottom_Press.Disable();
Top_Press.Disable();

SUPER^.Aborting();
END_METHOD

METHOD PROTECTED Clearing
VAR_INPUT
END_VAR
// CASE SequenceState OF
//     0:
//         NoStateTasksToComplete := FALSE;
//         SequenceState          := SequenceState + 10;
// 
//         //Trace('SequenceState: 10 - Initial state tasks set, moving to next state'); // Log initial state setup
//     10:
//         // Enable here
//         //         Bottom_Press_Hydro.Relax();
//         //         Top_Press_Hydro.Relax();
//         SequenceState := SequenceState + 10;
// 
//         //Trace('SequenceState: 20 - Main and Aux press hydraulics relaxed'); // Log hydraulic relaxation
//     20:
//         StateTasksComplete := TRUE;
// 
//     //Trace('StateTasksComplete: TRUE - State tasks completed'); // Log state tasks completion
// END_CASE

SUPER^.Clearing();
END_METHOD

METHOD PROTECTED Holding
VAR_INPUT
END_VAR
// CASE _CurrentMode OF
// =================================PRODUCTION MODE==================================
//     E_PMLUnitMode.ePMLUnitMode_Production:
//         CASE SequenceState OF
//             0:
//                 NoStateTasksToComplete := FALSE;
//                 SequenceState          := SequenceState + 10;
// 
//                 //Trace('SequenceState: 10 - Initial state tasks set, moving to next state'); // Log initial state setup
//             10:
//                 //                 Bottom_Press_Hydro.Relax();
//                 //                 Top_Press_Hydro.Relax();
//                 Bottom_Press.Stop();
//                 Top_Press.Stop();
// 
//                 IF Bottom_Press.Stopped AND Top_Press.Stopped THEN
//                     SequenceState := SequenceState + 10;
//                     //Trace('SequenceState: 20 - Both presses stopped'); // Log state transition when both presses are stopped
//                 END_IF
// 
//             20:
//                 // Disable here
//                 Bottom_Press.Disable();
//                 Top_Press.Disable();
//                 //Trace('SequenceState: 20 - Both presses disabled'); // Log presses disabled state
// 
//                 // Check not enabled here
//                 IF (NOT Bottom_Press.Enabled) AND (NOT Top_Press.Enabled) THEN
//                     SequenceState := SequenceState + 10;
//                     //Trace('SequenceState: 30 - Both presses not enabled'); // Log state transition when both presses are not enabled
//                 END_IF
// 
//             30:
//                 StateTasksComplete := TRUE;
// 
//             //Trace('StateTasksComplete: TRUE - State tasks completed'); // Log state tasks completion
//         END_CASE
// 
//         SUPER^.Holding();
// 
//     E_PMLUnitMode.ePMLUnitMode_Maintenance, E_PMLUnitMode.ePMLUnitMode_Manual:
//         SUPER^.Holding();
// END_CASE

Bottom_Press.Stop();
Top_Press.Stop();

SUPER^.Holding();
END_METHOD

METHOD PROTECTED Starting
VAR_INPUT
END_VAR
CASE DescendantSequenceState OF
    0:
        IF MotorsInit() THEN
            DescendantSequenceState := 10;
        END_IF

    10:
        Bottom_Press.MoveAbsolute(Position := BottomPressRecipe.OpenPosition, TRUE);
        Top_Press.MoveAbsolute(Position := TopPressRecipe.OpenPosition, TRUE);
        DescendantSequenceState := 15;

    15:
        IF TopPressRecipe.AtTop AND NOT Top_Press.Busy AND BottomPressRecipe.AtTop AND NOT Bottom_Press.Busy THEN
            //servo in position
            DescendantSequenceState := 20;
        END_IF

    20:
        _NailplateCountData_Ready  := FALSE;
        _NailplateCountData_Sent   := FALSE;
        _DoublePickData_Sent       := FALSE;
        _DoublePickData_Ready      := FALSE;
        BottomPressRecipe.SubState := 0;
        TopPressRecipe.SubState    := 0;
        BottomPressRecipe.State    := E_RamState.rsINIT;
        TopPressRecipe.State       := E_RamState.rsINIT;
        DetailIndex                := 1;

        Detail_Step := PRESS_INIT;
        SUPER^.Starting();
END_CASE
END_METHOD

METHOD PROTECTED Stopping
VAR_INPUT
END_VAR
// CASE SequenceState OF
//     0:
//         NoStateTasksToComplete := FALSE;
//         SequenceState          := SequenceState + 10;
// 
//         //Trace('SequenceState: 10 - Initial state tasks set, moving to next state'); // Log initial state setup
//     10:
//         //         Cooler.Cool := FALSE;
//         //         Bottom_Press_Hydro.Relax();
//         //         Top_Press_Hydro.Relax();
//         Bottom_Press.Stop();
//         Top_Press.Stop();
// 
//         //Trace('SequenceState: 10 - Cooler off, hydraulics relaxed, presses stopping'); // Log cooler, hydraulics, and press stop commands
//         IF Bottom_Press.Stopped AND Top_Press.Stopped THEN
//             SequenceState := SequenceState + 10;
//             //Trace('SequenceState: 20 - Both presses stopped'); // Log state transition when both presses are stopped
//         END_IF
// 
//     20:
//         // Disable here
//         Bottom_Press.Disable();
//         Top_Press.Disable();
//         //Trace('SequenceState: 20 - Both presses disabled'); // Log presses disabled state
// 
//         // Check not enabled here
//         IF (NOT Bottom_Press.Enabled) AND (NOT Top_Press.Enabled) THEN
//             SequenceState := SequenceState + 10;
//             //Trace('SequenceState: 30 - Both presses not enabled'); // Log state transition when both presses are not enabled
//         END_IF
// 
//     30:
//         StateTasksComplete := TRUE;
// 
//     //Trace('StateTasksComplete: TRUE - State tasks completed'); // Log state tasks completion
// END_CASE

Bottom_Press.Stop();
Top_Press.Stop();

SUPER^.Stopping();
END_METHOD

METHOD PROTECTED Suspending
VAR_INPUT
END_VAR
// CASE SequenceState OF
//     0:
//         NoStateTasksToComplete := FALSE;
//         SequenceState          := SequenceState + 10;
// 
//         //Trace('SequenceState: 10 - Initial state tasks set, moving to next state'); // Log initial state setup
//     10:
//         //         Bottom_Press_Hydro.Relax();
//         //         Top_Press_Hydro.Relax();
//         Bottom_Press.Stop();
//         Top_Press.Stop();
// 
//         //Trace('SequenceState: 10 - Hydraulics relaxed, presses stopping'); // Log hydraulics relaxation and presses stopping
//         IF Bottom_Press.Stopped AND Top_Press.Stopped THEN
//             SequenceState := SequenceState + 10;
//             //Trace('SequenceState: 20 - Both presses stopped'); // Log state transition when both presses are stopped
//         END_IF
// 
//     20:
//         // Disable here
//         Bottom_Press.Disable();
//         Top_Press.Disable();
//         //Trace('SequenceState: 20 - Both presses disabled'); // Log presses disabled state
// 
//         // Check not enabled here
//         IF (NOT Bottom_Press.Enabled) AND (NOT Top_Press.Enabled) THEN
//             SequenceState := SequenceState + 10;
//             //Trace('SequenceState: 30 - Both presses not enabled'); // Log state transition when both presses are not enabled
//         END_IF
// 
//     30:
//         StateTasksComplete := TRUE;
// 
//     //Trace('StateTasksComplete: TRUE - State tasks completed'); // Log state tasks completion
// END_CASE

Bottom_Press.Stop();
Top_Press.Stop();

SUPER^.Suspending();
END_METHOD

METHOD PROTECTED Unholding
VAR_INPUT
END_VAR
// CASE _CurrentMode OF
//     //=================================PRODUCTION MODE==================================
//     E_PMLUnitMode.ePMLUnitMode_Production:
//         CASE SequenceState OF
//             0:
//                 NoStateTasksToComplete := FALSE;
//                 Bottom_Press.Enable();
//                 Top_Press.Enable();
// 
//                 //Trace('SequenceState: 0 - Both presses enabled'); // Log enabling of presses
//                 // Check enabled here
//                 IF Bottom_Press.Enabled AND Top_Press.Enabled THEN
//                     SequenceState := 50; // Skipping movement on unholding
//                     //Trace('SequenceState: 50 - Skipping movement, both presses enabled'); // Log state transition when both presses are enabled
//                 END_IF
// 
//             10:
//                 Bottom_Press.Velocity     := BottomPressRecipe.Axis.Velocity;
//                 Bottom_Press.Acceleration := BottomPressRecipe.Axis.Acceleration;
//                 Bottom_Press.MoveAbsolute(Position := BottomPressRecipe.OpenPosition, TRUE);
//                 SequenceState := SequenceState + 10;
// 
//                 //Trace('SequenceState: 20 - Main press moving to open position'); // Log state transition and main press movement
//             20:
//                 IF Bottom_Press.InPosition AND NOT Bottom_Press.Busy THEN
//                     SequenceState := SequenceState + 10;
//                     //Trace('SequenceState: 30 - Main press in position'); // Log state transition when main press is in position
//                 END_IF
// 
//             30:
//                 Top_Press.Velocity     := TopPressRecipe.Axis.Velocity;
//                 Top_Press.Acceleration := TopPressRecipe.Axis.Acceleration;
//                 Top_Press.MoveAbsolute(Position := TopPressRecipe.OpenPosition, TRUE);
//                 SequenceState := SequenceState + 10;
// 
//                 //Trace('SequenceState: 40 - Aux press moving to open position'); // Log state transition and aux press movement
//             40:
//                 IF Top_Press.InPosition AND NOT Top_Press.Busy THEN
//                     SequenceState := SequenceState + 10;
//                     //Trace('SequenceState: 50 - Aux press in position'); // Log state transition when aux press is in position
//                 END_IF
// 
//             50:
//                 StateTasksComplete := TRUE;
//                 //Trace('StateTasksComplete: TRUE - State tasks completed'); // Log state tasks completion
//                 TopPressRecipe.SubState    := 0;
//                 BottomPressRecipe.SubState := 0;
//         END_CASE
// 
//         SUPER^.Unholding();
// 
//     E_PMLUnitMode.ePMLUnitMode_Maintenance, E_PMLUnitMode.ePMLUnitMode_Manual:
//         SUPER^.Unholding();
// END_CASE

TopPressRecipe.SubState    := 0;
BottomPressRecipe.SubState := 0;

SUPER^.Unholding();
END_METHOD

METHOD PROTECTED Unsuspending
VAR_INPUT
END_VAR
// CASE _CurrentMode OF
//     //=================================PRODUCTION MODE==================================
//     E_PMLUnitMode.ePMLUnitMode_Production, E_PMLUnitMode.ePMLUnitMode_Manual:
//         CASE SequenceState OF
//             0:
//                 NoStateTasksToComplete := FALSE;
//                 Bottom_Press.Enable();
//                 Top_Press.Enable();
// 
//                 //Trace('SequenceState: 0 - Both presses enabled'); // Log enabling of presses
//                 // Check enabled here
//                 IF Bottom_Press.Enabled AND Top_Press.Enabled THEN
//                     SequenceState := 50; // Skipping movement on unsuspending
//                     //Trace('SequenceState: 50 - Skipping movement, both presses enabled'); // Log state transition when both presses are enabled
//                 END_IF
// 
//             10:
//                 Bottom_Press.Velocity     := BottomPressRecipe.Axis.Velocity;
//                 Bottom_Press.Acceleration := BottomPressRecipe.Axis.Acceleration;
//                 Bottom_Press.MoveAbsolute(Position := BottomPressRecipe.OpenPosition, TRUE);
//                 SequenceState := SequenceState + 10;
// 
//                 //Trace('SequenceState: 10 - Main press moving to open position'); // Log state transition and main press movement
//             20:
//                 IF Bottom_Press.InPosition AND NOT Bottom_Press.Busy THEN
//                     SequenceState := SequenceState + 10;
//                     //Trace('SequenceState: 20 - Main press in position'); // Log state transition when main press is in position
//                 END_IF
// 
//             30:
//                 Top_Press.Velocity     := TopPressRecipe.Axis.Velocity;
//                 Top_Press.Acceleration := TopPressRecipe.Axis.Acceleration;
//                 Top_Press.MoveAbsolute(Position := TopPressRecipe.OpenPosition, TRUE);
//                 SequenceState := SequenceState + 10;
// 
//                 //Trace('SequenceState: 30 - Aux press moving to open position'); // Log state transition and aux press movement
//             40:
//                 IF Top_Press.InPosition AND NOT Top_Press.Busy THEN
//                     SequenceState := SequenceState + 10;
//                     //Trace('SequenceState: 40 - Aux press in position'); // Log state transition when aux press is in position
//                 END_IF
// 
//             50:
//                 StateTasksComplete := TRUE;
// 
//             //Trace('StateTasksComplete: TRUE - State tasks completed'); // Log state tasks completion
//         END_CASE
// 
//         //=================================MAINTENANCE MODE==================================
//     E_PMLUnitMode.ePMLUnitMode_Maintenance:
//         ;
// END_CASE

TopPressRecipe.SubState    := 0;
BottomPressRecipe.SubState := 0;

SUPER^.Unsuspending();
END_METHOD

METHOD AssemblyEnd : BOOL
END_METHOD

METHOD AssemblyStart : BOOL
END_METHOD

METHOD ExecuteDetail : BOOL
VAR_INPUT
    DetailToRun : UDINT;
END_VAR

VAR_INST
    Previous_State : E_Press_States;
END_VAR
ExecuteDetail := FALSE;

CASE Detail_Step OF
    PRESS_INIT:
        IF Plates.Plates[DetailToRun].TopOrBottom = 'Top' THEN
            TopPressRecipe.State    := E_RamState.rsFULL_RETRACT;
            BottomPressRecipe.State := E_RamState.rsEXTEND_TO_BACKER;

            IF TopPressRecipe.State_Response = E_RamState.rsFULL_RETRACT AND BottomPressRecipe.State_Response = E_RamState.rsEXTEND_TO_BACKER THEN
                Detail_Step := NP_READY_TO_PLACE_WS;
            END_IF
        ELSIF Plates.Plates[DetailToRun].TopOrBottom = 'Bottom' THEN
            TopPressRecipe.State    := E_RamState.rsEXTEND_TO_BACKER;
            BottomPressRecipe.State := E_RamState.rsFULL_RETRACT;

            IF TopPressRecipe.State_Response = E_RamState.rsEXTEND_TO_BACKER AND BottomPressRecipe.State_Response = E_RamState.rsFULL_RETRACT THEN
                Detail_Step := NP_READY_TO_PLACE_WS;
            END_IF
        END_IF

    NP_READY_TO_PLACE_WS:
        IF WaitSync_Handler(E_WaitSync.NAILPLATE_READY_TO_PLACE) THEN
            Detail_Step := ROBOT_PERMISSION_REQUEST;
        END_IF

    ROBOT_PERMISSION_REQUEST:
        _PressRobotPermissionToEnter.Request := TRUE;

        IF _PressRobotPermissionToEnter.Permission THEN
            Detail_Step := ROBOT_PERMISSION_GRANTED_WS;
        END_IF

    ROBOT_PERMISSION_GRANTED_WS:
        IF WaitSync_Handler(E_WaitSync.PRESS_ROBOT_PERMISSION_GRANTED) THEN
            Detail_Step := NP_PLACED_WS;
        END_IF

    NP_PLACED_WS:
        IF WaitSync_Handler(E_WaitSync.NAILPLATE_PLACED) THEN
            Detail_Step := NP_PREP_POS;
        END_IF

    NP_PREP_POS:
        IF Plates.Plates[DetailToRun].TopOrBottom = 'Top' THEN
            TopPressRecipe.State := E_RamState.rsEXTEND_TO_CLOSED_PREP;

            IF TopPressRecipe.State_Response = E_RamState.rsEXTEND_TO_CLOSED_PREP THEN
                Detail_Step := READY_FOR_BOARD_WS;
            END_IF
        ELSIF Plates.Plates[DetailToRun].TopOrBottom = 'Bottom' THEN
            BottomPressRecipe.State := E_RamState.rsEXTEND_TO_CLOSED_PREP;

            IF BottomPressRecipe.State_Response = E_RamState.rsEXTEND_TO_CLOSED_PREP THEN
                Detail_Step := READY_FOR_BOARD_WS;
            END_IF
        END_IF

    READY_FOR_BOARD_WS:
        _PressRobotPermissionToEnter.Request := FALSE;

        IF WaitSync_Handler(E_WaitSync.CARRIAGE2_PRESS_READY_FOR_BOARD) THEN
            Detail_Step := BOARD_IN_POSITION_WS;
        END_IF

    BOARD_IN_POSITION_WS:
        IF WaitSync_Handler(E_WaitSync.CARRIAGE2_PRESS_BOARD_IN_POSITION) THEN
            Detail_Step := PRESSING_NAILPLATE;
        END_IF

    PRESSING_NAILPLATE:
        IF Plates.Plates[DetailToRun].TopOrBottom = 'Top' THEN
            TopPressRecipe.State    := E_RamState.rsEXTEND_TO_PRESSURE;
            BottomPressRecipe.State := E_RamState.rsEXTEND_TO_CLOSED;

            IF TopPressRecipe.State_Response = E_RamState.rsEXTEND_TO_PRESSURE AND BottomPressRecipe.State_Response = E_RamState.rsEXTEND_TO_CLOSED
            THEN
                Detail_Step := RETRACTING_FOR_INDEX;
            END_IF
        ELSIF Plates.Plates[DetailToRun].TopOrBottom = 'Bottom' THEN
            BottomPressRecipe.State := E_RamState.rsEXTEND_TO_PRESSURE;
            TopPressRecipe.State    := E_RamState.rsEXTEND_TO_CLOSED;

            IF BottomPressRecipe.State_Response = E_RamState.rsEXTEND_TO_PRESSURE AND TopPressRecipe.State_Response = E_RamState.rsEXTEND_TO_CLOSED
            THEN
                Detail_Step := RETRACTING_FOR_INDEX;
            END_IF
        END_IF

    RETRACTING_FOR_INDEX:
        TopPressRecipe.State    := E_RamState.rsRETRACT_FOR_INDEX;
        BottomPressRecipe.State := E_RamState.rsRETRACT_FOR_INDEX;

        IF TopPressRecipe.State_Response = E_RamState.rsRETRACT_FOR_INDEX AND BottomPressRecipe.State_Response = E_RamState.rsRETRACT_FOR_INDEX THEN
            Detail_Step := NP_DONE_WS;
        END_IF

    NP_DONE_WS:
        IF WaitSync_Handler(E_WaitSync.CARRIAGE2_PRESS_NAILPLATE_DONE) THEN
            ExecuteDetail := TRUE;
            Detail_Step   := PRESS_INIT;
        END_IF

END_CASE

IF Detail_Step <> Previous_State THEN
    Trace(CONCAT('Press StepDetail state change to: ', TO_STRING(Detail_Step)));
END_IF

Previous_State := Detail_Step;
END_METHOD

METHOD ExecuteStep : BOOL
VAR_INPUT
    Step : ST_CSV_Step;
END_VAR

VAR
    EmptyPlates : ST_Plates;
END_VAR
ExecuteStep := FALSE;

CASE Step.seqName OF

    E_CommandName.BoardInfo:
		BoardInfoParse(Step := Step, StepOut := _BoardDataToPass);

//         _NailplateCountDataToPass := STRING_TO_UDINT(Step.Details[1].Datas[6]);
//         _BoardLength              := STRING_TO_LREAL(Step.Details[1].Datas[5]);

        IF _BoardDataToPass.TotalPlates = 0 THEN
            IF _NailplateCountData_Sent = FALSE THEN
                _NailplateCountData_Sent := WaitSync_Handler(E_WaitSync.HANDOFF2_PRESS_TOTAL_NP_COUNT);
           ELSE
                IF WaitSync_Handler(E_WaitSync.HANDOFF2_PRESS_DOUBLE_PICK) THEN
                    ExecuteStep               := TRUE;
                    _NailplateCountData_Ready := FALSE;
                    _NailplateCountData_Sent  := FALSE;
                    _DoublePickData_Sent      := FALSE;
                    _DoublePickData_Ready     := FALSE;
                END_IF
            END_IF
        ELSE
            _DoublePickData_Sent  := FALSE;
            _DoublePickData_Ready := FALSE;

            IF WaitSync_Handler(E_WaitSync.HANDOFF2_PRESS_TOTAL_NP_COUNT) THEN
                ExecuteStep := TRUE;
// 		 		Trace(CONCAT('HANDOFF2_PRESS_TOTAL_NP_COUNT done for board:  ',Concat(_BoardDataToPass.BoardID,CONCAT(' -> ',INT_TO_STRING(_BoardDataToPass.BoardNumber)))));
            END_IF
        END_IF
		Plates := EmptyPlates;
    E_CommandName.NailPlate:
        NailPlateParse(Step, Plates);
        _DoublePickDataToPass := DoublePickNailPlatePosCheck(Plates, _BoardDataToPass.BoardLength);

        IF _DoublePickData_Sent = FALSE THEN
            _DoublePickData_Sent := WaitSync_Handler(E_WaitSync.HANDOFF2_PRESS_DOUBLE_PICK);
        ELSE
            _NailplateDataToPass      := Plates.Plates[DetailIndex];
            IF ExecuteDetail(DetailIndex) THEN
                DetailIndex := DetailIndex + 1;
            END_IF


            IF DetailIndex > Step.DetailCount THEN
                DetailIndex               := 1;
                ExecuteStep               := TRUE;
                _DoublePickData_Sent      := FALSE;
                _DoublePickData_Ready     := FALSE;
                _NailplateCountData_Ready := FALSE;
                _NailplateCountData_Sent  := FALSE;
           END_IF
        END_IF

ELSE
    ExecuteStep := TRUE;
END_CASE
END_METHOD

METHOD PROTECTED Execute
VAR_INPUT
END_VAR

VAR_INST
    dwellTime         : TON;
    EDGEPOS_InitCycle : R_TRIG;
END_VAR

VAR
    TestCycle : BOOL := FALSE;
END_VAR
CASE _CurrentMode OF
    //=================================PRODUCTION MODE==================================
    E_PMLUnitMode.ePMLUnitMode_Production:

        PressLogic(Bottom_Press, BottomPressRecipe);
        PressLogic(Top_Press, TopPressRecipe);

        //=================================MAINTENANCE & MANUAL MODE==================================        
    E_PMLUnitMode.ePMLUnitMode_Maintenance, E_PMLUnitMode.ePMLUnitMode_Manual:
        ; // No specific actions, just log the mode

    //Trace('Mode: Maintenance or Manual - No actions taken'); // Log maintenance or manual mode entry
END_CASE

SUPER^.Execute();
END_METHOD

METHOD DoublePickNailPlatePosCheck : BOOL
VAR_INPUT
    PlateInfo : REFERENCE TO ST_Plates;
    Length    : REFERENCE TO REAL;
END_VAR

VAR
    MaxNailplatePos : lreal;
END_VAR
DoublePickNailPlatePosCheck := FALSE;

FOR i := 1 TO MAX_NUMBER_OF_PLATES DO
    MaxNailplatePos := MAX(PlateInfo.Plates[i].PlatePlaceX, MaxNailplatePos);
END_FOR

IF Length > Global.DOUBLEPICK_MIN_LENGTH AND (Length - MaxNailplatePos) < Global.DOUBLEPICK_MIN_LENGTH AND MaxNailplatePos > 1000 THEN
    DoublePickNailPlatePosCheck := TRUE;
END_IF
END_METHOD

METHOD HMIControl
VAR_INPUT
END_VAR

VAR_INST
    PowerOnCommand_Top     : BOOL;
    PowerOffCommand_Top    : BOOL;
    PowerOnCommand_Bottom  : BOOL;
    PowerOffCommand_Bottom : BOOL;
END_VAR
Top_PressCmds_Extra.Temp_R_Trig[1](CLK := Top_PressCmds_Extra.MotorCmd[1]);

PowerOnCommand_Top := Top_PressCmds_Extra.Temp_R_Trig[1].Q AND PowerOnCommand_Top = FALSE;

IF PowerOnCommand_Top THEN
    IF Top_Press.Enable() THEN
        PowerOnCommand_Top := FALSE;
    END_IF
END_IF

Top_PressCmds_Extra.Temp_R_Trig[2](CLK := Top_PressCmds_Extra.MotorCmd[2]);

PowerOffCommand_Top := Top_PressCmds_Extra.Temp_R_Trig[2].Q AND PowerOffCommand_Top = FALSE;

IF PowerOffCommand_Top THEN
    IF Top_Press.Disable() THEN
        PowerOffCommand_Top := FALSE;
    END_IF
END_IF

Bottom_PressCmds_Extra.Temp_R_Trig[1](CLK := Bottom_PressCmds_Extra.MotorCmd[1]);

PowerOnCommand_Bottom := Bottom_PressCmds_Extra.Temp_R_Trig[1].Q AND PowerOnCommand_Bottom = FALSE;

IF PowerOnCommand_Bottom THEN
    IF Bottom_Press.Enable() THEN
        PowerOnCommand_Bottom := FALSE;
    END_IF
END_IF

Bottom_PressCmds_Extra.Temp_R_Trig[2](CLK := Bottom_PressCmds_Extra.MotorCmd[2]);

PowerOffCommand_Bottom := Bottom_PressCmds_Extra.Temp_R_Trig[2].Q AND PowerOffCommand_Bottom = FALSE;

IF PowerOffCommand_Bottom THEN
    IF Bottom_Press.Disable() THEN
        PowerOffCommand_Bottom := FALSE;
    END_IF
END_IF
END_METHOD

//! @summary Basic module initialization logic
METHOD PROTECTED Initialize : BOOL;
VAR
    i                        : UDINT;
    varInfo                  : __SYSTEM.VAR_INFO;
    AllSubUnitsInitialized   : BOOL := TRUE;
    AllComponentsInitialized : BOOL := TRUE;
END_VAR

//! @description This method is called by <c>CyclicLogic()</c> as required
Initialize := FALSE;

CASE DescendantSequenceState OF
    0:
        RegisterComponent(Top_Press);
        RegisterComponent(Bottom_Press);

        _LogModeChanges         := FALSE;
        _LogStateChanges        := FALSE;
        DescendantSequenceState := DescendantSequenceState + 10;

    10:
        //Setup Custom modes here

        (*CustomModes(eMode                          :=,
                    sName                          :=,
                    bDisableClearing               :=,
                    bDisableStarting               :=,
                    bDisableSuspended              :=,
                    bDisableStopping               :=,
                    bDisableAborting               :=,
                    bDisableHolding                :=,
                    bDisableHeld                   :=,
                    bDisableUnholding              :=,
                    bDisableSuspending             :=,
                    bDisableUnsuspending           :=,
                    bDisableResetting              :=,
                    bDisableIdle                   :=,
                    bDisableCompleting             :=,
                    bDisableComplete               :=,
                    bEnableUnitModeChangeStopped   :=,
                    bEnableUnitModeChangeIdle      :=,
                    bEnableUnitModeChangeSuspended :=,
                    bEnableUnitModeChangeExecute   :=,
                    bEnableUnitModeChangeAborted   :=,
                    bEnableUnitModeChangeHeld      :=,
                    bEnableUnitModeChangeComplete  :=,
                    bError                         =>,
                    nErrorId                       =>);*)

        DescendantSequenceState := DescendantSequenceState + 10;

    20:
        //Copy Mode names

        FOR i := 1 TO 3 DO
            ModeNames[i] := F_UnitModeToString(UDINT_TO_DINT(i));
        END_FOR

        RegisterExternalController(Controller := fbControlSourceHMI);
        fbControlSourceHMI.CyclicLogic();
        DescendantSequenceState := DescendantSequenceState + 10;

    30:
        //Call the Super

        IF SUPER^.Initialize() THEN
            DescendantSequenceState := DescendantSequenceState + 10;
        END_IF

    40:
        Initialize := TRUE;
END_CASE
END_METHOD

METHOD MotorsInit : BOOL
VAR_INPUT
END_VAR
MotorsInit := FALSE;

IF _InSimulation THEN
    IF MotorResetAndEnable(Top_Press) AND MotorResetAndEnable(Bottom_Press) THEN
        MotorsInit := TRUE;
    END_IF
ELSE
    IF MotorResetAndEnable(Top_Press) AND MotorResetAndEnable(Bottom_Press) THEN
        MotorsInit := TRUE;
    END_IF
END_IF
END_METHOD

METHOD PressLogic : BOOL
VAR_INPUT
    PressMotor : REFERENCE TO FB_Component_BasicSlaveAxis_SoE;
    Recipe     : REFERENCE TO ST_PressRecipe;
END_VAR

VAR
    TorqueMoveEnabled : BOOL := FALSE;
END_VAR
//reset response

Recipe.State_Response := E_RamState.rsUNDEFINED;

CASE Recipe.State OF
    E_RamState.rsIDLE, E_RamState.rsINIT:

        PressMotor.Velocity     := Recipe.Axis.Velocity;
        PressMotor.Acceleration := Recipe.Axis.Acceleration;

        Recipe.State_Response := Recipe.State;

    E_RamState.rsFULL_RETRACT:

        CASE Recipe.SubState OF
            0:
                PressMotor.MoveAbsolute(Position := Recipe.OpenPosition, TRUE);
                Recipe.SubState := Recipe.SubState + 1;

            1:
                //wait for servo to get into position

                IF Recipe.AtTop AND NOT PressMotor.Busy THEN
                    //servo in position

                    Recipe.State_Response := Recipe.State;
                END_IF
        END_CASE

    E_RamState.rsFULL_EXTEND:
        ;

    E_RamState.rsEXTEND_TO_BACKER:
        CASE Recipe.SubState OF
            0:
                PressMotor.MoveAbsolute(Position := Recipe.BackerPosition, TRUE);
                Recipe.SubState := Recipe.SubState + 1;

            1:
                //wait for servo to get into position

                IF Recipe.AtWork AND NOT PressMotor.Busy THEN
                    //servo in position

                    Recipe.State_Response := Recipe.State;
                END_IF
        END_CASE

    E_RamState.rsEXTEND_TO_CLOSED:
        CASE Recipe.SubState OF
            0:
                PressMotor.MoveAbsolute(Position := Recipe.ClosedPosition, TRUE);
                Recipe.SubState := Recipe.SubState + 1;

            1:
                //wait for servo to get into position

                IF PressMotor.InPosition AND NOT PressMotor.Busy THEN
                    //servo in position

                    Recipe.State_Response := Recipe.State;
                END_IF
        END_CASE

        // this state will start movement to a closed prep position after nailplate is placed.  movement will be overrided if next movement is hit before this one finishes
    E_RamState.rsEXTEND_TO_CLOSED_PREP:
        CASE Recipe.SubState OF
            0:
                PressMotor.MoveAbsolute(Position := Recipe.ClosedPosition - 70, TRUE);
                Recipe.SubState := Recipe.SubState + 1;

            1:
                //wait for servo to get into position

                IF PressMotor.Busy THEN
                    //servo in position

                    Recipe.State_Response := Recipe.State;
                END_IF
        END_CASE

    E_RamState.rsEXTEND_TO_PRESSURE:
        CASE Recipe.SubState OF
            0:
                IF RobotClearOfPress THEN
                    IF TorqueMoveEnabled THEN
                        Recipe.SubState := 10;
                    ELSE
                        Recipe.SubState := 20;

                    END_IF
                END_IF

            10:
                Recipe.TorqueOptions.EnableManualTorqueStartValue := TRUE;
                Recipe.TorqueOptions.ManualTorqueStartValue       := PressMotor.Axis.NcToPlc.ActTorque;
                Recipe.Execute_TorqueMove                         := FALSE;

                Recipe.TorqueControl.Torque := Recipe.Axis.Torque;
                Trace('Press Motor Torque Command High');

                IF ABS(PressMotor.Axis.NcToPlc.ActTorque - Recipe.TorqueControl.Torque) < 0.5 AND PressMotor.Axis.NcToPlc.ActVelo < 0.5 THEN
                    Recipe.SubState           := 50;
                    Recipe.Execute_TorqueMove := FALSE;
                END_IF

            20:
                PressMotor.MoveAbsolute(Position := Recipe.ClosedPosition + 4, TRUE);
                Recipe.SubState := 21;

            21:
                //wait for servo to get into position

                IF Recipe.AtWork AND NOT PressMotor.Busy THEN
                    //servo in position

                    Recipe.SubState := 50;
                END_IF

            50:
                IF PressMotor.ActualVelocity < 1 THEN
                    PressMotor.Stop();

                    IF PressMotor.Stopped THEN
                        Recipe.State_Response := Recipe.State;
                    END_IF
                END_IF
        END_CASE

    E_RamState.rsRETRACT_FOR_INDEX:
        CASE Recipe.SubState OF
            0:
                PressMotor.MoveAbsolute(Position := Recipe.ClosedPosition - 10, TRUE);
                Recipe.SubState := Recipe.SubState + 1;

            1:
                //wait for servo to get into position

                IF PressMotor.ActualPosition < Recipe.ClosedPosition THEN
                    //servo in position

                    Recipe.SubState := Recipe.SubState + 1;
                END_IF

            2:

                Recipe.State_Response := Recipe.State;

        END_CASE

    E_RamState.rsERROR:
        PressMotor.Stop();

END_CASE

Recipe.TorqueControl(Axis              := PressMotor.Axis,
                     Execute           := Recipe.Execute_TorqueMove,
                     TorqueRamp        := 50,
                     VelocityLimitHigh := Recipe.Axis.Velocity,
                     VelocityLimitLow  := -Recipe.Axis.Velocity,
                     Options           := Recipe.TorqueOptions);

//if we have changed states, make sure to reset sub step

IF Recipe.State <> Recipe.State_Previous THEN
    Recipe.SubState := 0;
    Trace(CONCAT('RamState changed state to: ', TO_STRING(Recipe.State)));
END_IF

Recipe.State_Previous := Recipe.State;
END_METHOD

PROPERTY BoardDataToPass : ST_BoardInfo
GET
BoardDataToPass := _BoardDataToPass;
END_GET
END_PROPERTY

PROPERTY DoublePickData_Ready : bool
GET
DoublePickData_Ready := _DoublePickData_Ready;
END_GET
END_PROPERTY

PROPERTY DoublePickData_Sent : bool
GET
DoublePickData_Sent := _DoublePickData_Sent;
END_GET
SET
_DoublePickData_Sent := DoublePickData_Sent;
END_SET
END_PROPERTY

PROPERTY DoublePickDataToPass : bool
GET
DoublePickDataToPass := _DoublePickDataToPass;
END_GET
END_PROPERTY

PROPERTY NailplateCountData_Ready : bool
GET
NailplateCountData_Ready := _NailplateCountData_Ready;
END_GET
END_PROPERTY

PROPERTY NailplateCountData_Sent : bool
GET
NailplateCountData_Sent := _NailplateCountData_Sent;
END_GET
SET
_NailplateCountData_Sent := NailplateCountData_Sent;
END_SET
END_PROPERTY

PROPERTY NailplateDataToPass : ST_PlateInfo
GET
NailplateDataToPass := _NailplateDataToPass;
END_GET
END_PROPERTY

PROPERTY PressRobotPermissionToEnter : REFERENCE TO ST_MediatorInterface
GET
PressRobotPermissionToEnter REF= _PressRobotPermissionToEnter;
END_GET
SET
_PressRobotPermissionToEnter := PressRobotPermissionToEnter;
END_SET
END_PROPERTY

END_FUNCTION_BLOCK

// Machine/EquipmentModules/Functional Layer/FB_Robot
FUNCTION_BLOCK FB_Robot EXTENDS FB_EquipmentModule_SR
VAR
    // Sub module definitions here

    // List of sub modules

    ipSubModules_Init : ARRAY[1..Parameters_PackML_Base.MAX_NO_OF_SUBMODULES] OF I_PackML_BaseModule := [];

    // Component definitions here

    Robot : FB_Component_Robot := (Name := 'Robot');

END_VAR

VAR

    //Properties
    DetailIndex : UDINT := 1;

    Handshake_Step : DINT;

    _DryRun : BOOL;

END_VAR

METHOD CyclicLogic
VAR_INPUT
END_VAR

VAR

END_VAR
IF NOT _InitComplete THEN
    _InitComplete := Initialize();
    RETURN;
END_IF

//SimulationOn();

// transfer var from EM to COMP

// IF _Name = 'Robot 1' THEN

//     Robot.RobotType := 'Handling';

// ELSIF _Name = 'Robot 2' OR _Name = 'Robot 3' THEN

//     Robot.RobotType := 'Fastening';

// END_IF

SUPER^.CyclicLogic();
END_METHOD

METHOD CyclicLogicSimulation : BOOL
VAR_INPUT
END_VAR
END_METHOD

METHOD PROTECTED Aborting
VAR_INPUT
END_VAR
Handshake_Step                      := 0;
Robot.Handshake.OUT.Execute_Step    := FALSE;
Robot.Handshake.OUT.Execute_StepNum := 0;
DetailIndex                         := 1;

Super^.Aborting();
END_METHOD

METHOD PROTECTED Clearing
VAR_INPUT
END_VAR
Super^.Clearing();
END_METHOD

METHOD PROTECTED Completing
VAR_INPUT
END_VAR
Super^.Completing();
END_METHOD

METHOD PROTECTED Holding
VAR_INPUT
END_VAR
IF Robot.Handshake.IN.TaskRunning = FALSE THEN
    SUPER^.Holding();
END_IF
END_METHOD

METHOD PROTECTED Resetting
VAR_INPUT
END_VAR
// reset handshake step
Handshake_Step                      := 0;
Robot.Handshake.OUT.Execute_Step    := FALSE;
Robot.Handshake.OUT.Execute_StepNum := 0;
DetailIndex                         := 1;

Super^.Resetting();
END_METHOD

METHOD PROTECTED Starting
VAR_INPUT
END_VAR
Handshake_Step                      := 0;
Robot.Handshake.OUT.Execute_Step    := FALSE;
Robot.Handshake.OUT.Execute_StepNum := 0;
DetailIndex                         := 1;

Super^.Starting();
END_METHOD

METHOD PROTECTED Stopping
VAR_INPUT
END_VAR
Super^.Stopping();
END_METHOD

METHOD PROTECTED Suspending
VAR_INPUT
END_VAR
IF Robot.Handshake.IN.TaskRunning = FALSE THEN
    SUPER^.Suspending();
END_IF
END_METHOD

METHOD PROTECTED Unholding
VAR_INPUT
END_VAR
SUPER^.Unholding();
END_METHOD

METHOD PROTECTED Unsuspending
VAR_INPUT
END_VAR
IF Robot.Handshake.IN.TaskRunning OR _InSimulation OR _ForceHold THEN
    SUPER^.Unsuspending();
END_IF
END_METHOD

METHOD NailPlate : BOOL
VAR_INPUT
    Step : ST_CSV_Step;
END_VAR
// clear out array first
Robot.Clear_DataToSend();

// first entry is always step type
Robot.RecipeData_ToSend[1] := DINT_TO_USINT(E_CommandName.NailPlate);

// Robot.RecipeData_ToSend[2] := INT_TO_USINT(Plates[1].PlateNumber);
// 
// Robot.RecipeData_ToSend[3] := STRING_TO_USINT(Plates[1].PlateGauge);
// 
// Robot.RecipeData_ToSend[4] := LREAL_TO_USINT(TRUNC(Plates[1].PlateWidth * 10));
// 
// Robot.RecipeData_ToSend[5] := LREAL_TO_USINT(TRUNC(Plates[1].PlateHeight * 10));
// 
// Robot.RecipeData_ToSend[6] := LREAL_TO_USINT(TRUNC(Plates[1].PlatePlaceX * 10));
// 
// Robot.RecipeData_ToSend[7] := LREAL_TO_USINT(TRUNC(Plates[1].PlatePlaceY * 10));
// 
// Robot.RecipeData_ToSend[8] := LREAL_TO_USINT(TRUNC(Plates[1].PlatePlaceAngle * 10));
END_METHOD

METHOD PROTECTED Execute
VAR_INPUT
END_VAR
//  logic
WaitSync_Robot();

SubModuleMonitor();

SUPER^.Execute();
END_METHOD

METHOD ExtractNumFromString : DINT
VAR_INPUT
    InputString : STRING;
END_VAR

VAR
    NumberString : STRING     := ''; // Temporary string to collect digits
    Numbers      : STRING[10] := '0123456789'; // Temporary string to collect digits
    CurrentChar  : BYTE; // Current character being processed
    Result       : UDINT := 0; // Final extracted number as UDINT
    i            : INT   := 1; // String index
END_VAR
ExtractNumFromString := 0;
j                    := 0;

FOR i := 0 TO LEN(InputString) DO
    CurrentChar := InputString[i];

    // Check if the current character is a digit
    IF CurrentChar >= Numbers[0] AND CurrentChar <= Numbers[9] THEN
        NumberString[j] := CurrentChar;
        j               := j + 1;
    END_IF
END_FOR

// Check for a number at the end of the string
IF LEN(NumberString) > 0 THEN
    ExtractNumFromString := STRING_TO_DINT(NumberString); // Convert to UDINT
END_IF
END_METHOD

METHOD HMIControl
VAR_INPUT
END_VAR
END_METHOD

//! @summary Basic module initialization logic
METHOD PROTECTED Initialize : BOOL;
VAR
    i                        : UDINT;
    varInfo                  : __SYSTEM.VAR_INFO;
    AllSubUnitsInitialized   : BOOL := TRUE;
    AllComponentsInitialized : BOOL := TRUE;
END_VAR

//! @description This method is called by <c>CyclicLogic()</c> as required
Initialize := FALSE;

CASE DescendantSequenceState OF
    0:
        RegisterComponent(Robot);

        _LogModeChanges         := FALSE;
        _LogStateChanges        := FALSE;
        DescendantSequenceState := DescendantSequenceState + 10;

    10:
        //Setup Custom modes here

        (*CustomModes(eMode                          :=,
                    sName                          :=,
                    bDisableClearing               :=,
                    bDisableStarting               :=,
                    bDisableSuspended              :=,
                    bDisableStopping               :=,
                    bDisableAborting               :=,
                    bDisableHolding                :=,
                    bDisableHeld                   :=,
                    bDisableUnholding              :=,
                    bDisableSuspending             :=,
                    bDisableUnsuspending           :=,
                    bDisableResetting              :=,
                    bDisableIdle                   :=,
                    bDisableCompleting             :=,
                    bDisableComplete               :=,
                    bEnableUnitModeChangeStopped   :=,
                    bEnableUnitModeChangeIdle      :=,
                    bEnableUnitModeChangeSuspended :=,
                    bEnableUnitModeChangeExecute   :=,
                    bEnableUnitModeChangeAborted   :=,
                    bEnableUnitModeChangeHeld      :=,
                    bEnableUnitModeChangeComplete  :=,
                    bError                         =>,
                    nErrorId                       =>);*)

        DescendantSequenceState := DescendantSequenceState + 10;

    20:
        //Copy Mode names

        FOR i := 1 TO 3 DO
            ModeNames[i] := F_UnitModeToString(UDINT_TO_DINT(i));
        END_FOR

        RegisterExternalController(Controller := fbControlSourceHMI);
        fbControlSourceHMI.CyclicLogic();
        DescendantSequenceState := DescendantSequenceState + 10;

    30:
        //Call the Super

        IF SUPER^.Initialize() THEN
            DescendantSequenceState := DescendantSequenceState + 10;
        END_IF

    40:
        Initialize := TRUE;
END_CASE
END_METHOD

METHOD WaitSync_Robot : BOOL
VAR
END_VAR

VAR_INST
    State : UDINT;
END_VAR
CASE State OF
    0:
        IF Robot.Handshake.IN.SubStepNumber > E_WaitSync.EMPTY THEN
            State := 1;
        END_IF

    1:
        _RequestedWaitSync := Robot.Handshake.IN.SubStepNumber;

        IF _RequestedWaitSync = _ResponseWaitSync THEN
            State := 2;
        END_IF

    2:
        Robot.Handshake.OUT.SubStepResponse := _ResponseWaitSync;

        IF Robot.Handshake.IN.SubStepNumber = E_WaitSync.EMPTY THEN
            _RequestedWaitSync := Robot.Handshake.IN.SubStepNumber;

            IF _ResponseWaitSync = E_WaitSync.EMPTY THEN
                Robot.Handshake.OUT.SubStepResponse := E_WaitSync.EMPTY;
                State                               := 0;
            END_IF
        END_IF

END_CASE
END_METHOD

PROPERTY DryRun : BOOL
GET
DryRun := _DryRun;
END_GET
SET
_DryRun := DryRun;
END_SET
END_PROPERTY

PROPERTY OtherInputs : ARRAY[0..7] OF USINT
GET
OtherInputs := Robot.OtherInputs;
END_GET
END_PROPERTY

PROPERTY OtherOutputs : ARRAY[0..7] OF USINT
SET
Robot.OtherOutputs := OtherOutputs;
END_SET
END_PROPERTY

(*! @summary This method monitors <b>submodules</b> within this PackML module and initiates fault responses as required*)
METHOD PROTECTED SubModuleMonitor : BOOL
SUPER^.SubModuleMonitor();
END_METHOD

END_FUNCTION_BLOCK

// Machine/EquipmentModules/Functional Layer/FB_Robot_Outfeed
FUNCTION_BLOCK FB_Robot_Outfeed EXTENDS FB_Robot
VAR
    // Sub module definitions here

    _PickPlaceDataToPass : ST_PickPlace;
END_VAR

VAR

    PickPlaceData : ST_PickPlace;

END_VAR

METHOD CyclicLogic
VAR_INPUT
END_VAR

VAR

END_VAR
IF NOT _InitComplete THEN
    _InitComplete := Initialize();
    RETURN;
END_IF

SUPER^.CyclicLogic();

UI_MessageBox();
END_METHOD

METHOD CyclicLogicSimulation : BOOL
VAR_INPUT
END_VAR
END_METHOD

METHOD ExecuteDetail : BOOL
VAR_INPUT
    StepToRun : UDINT;
END_VAR
ExecuteDetail := FALSE;

CASE Handshake_Step OF
    0:
        Robot.Handshake.OUT.Execute_Step    := TRUE;
        Robot.Handshake.OUT.Execute_StepNum := UDINT_TO_UINT(StepToRun);

        IF Robot.Handshake.IN.Executing_Step = TRUE THEN
            Handshake_Step := 1;
        END_IF

    1:
        IF Robot.Handshake.IN.Executing_Step = FALSE AND Robot.Handshake.IN.StepComplete = TRUE THEN
            Handshake_Step := 2;
        END_IF

    2:
        Robot.Handshake.OUT.Execute_Step    := FALSE;
        Robot.Handshake.OUT.Execute_StepNum := 0;

        IF Robot.Handshake.IN.StepComplete = FALSE THEN
            ExecuteDetail  := TRUE;
            Handshake_Step := 0;
        END_IF

END_CASE
END_METHOD

METHOD PROTECTED ExecuteDetail_SIM : BOOL
VAR_INPUT
    StepToRun : UDINT;
    LineNum   : INT;
END_VAR

VAR_INST
    robotWS_State : E_AssemblyPickState;
END_VAR
CASE robotWS_State OF
    BOARD_READY_WS:
        IF WaitSync_Handler(E_WaitSync.PICK1_ASSEMBLY_BOARD_READY) THEN
            robotWS_State := OPEN_GRIPPERS_WS;
        END_IF

    OPEN_GRIPPERS_WS:
        IF WaitSync_Handler(E_WaitSync.PICK1_ASSEMBLY_OPEN_GRIPPERS) THEN
            robotWS_State := PICKING_BOARD_WS;
        END_IF

    PICKING_BOARD_WS:
        IF WaitSync_Handler(E_WaitSync.PICK1_ASSEMBLY_PICKING_BOARD) THEN
            robotWS_State := BOARD_CLEAR_WS;
        END_IF

    BOARD_CLEAR_WS:
        IF WaitSync_Handler(E_WaitSync.PICK1_ASSEMBLY_BOARD_CLEAR) THEN
            IF LineNum = 1 THEN
                robotWS_State := SIM_JIG2READYPLACE_WS;
            ELSE
                robotWS_State := SIM_JIG3READYPLACE_WS;
            END_IF
        END_IF

    SIM_JIG2READYPLACE_WS:
        IF WaitSync_Handler(E_WaitSync.OUTFEED_JIG2_PICKPLACE_READY) THEN
            robotWS_State := SIM_JIG2PLACEDONE_WS;
        END_IF

    SIM_JIG2PLACEDONE_WS:
        IF WaitSync_Handler(E_WaitSync.OUTFEED_JIG2_PICKPLACE_DONE) THEN
            robotWS_State := PICK_DONE;
        END_IF

    SIM_JIG3READYPLACE_WS:
        IF WaitSync_Handler(E_WaitSync.OUTFEED_JIG3_PICKPLACE_READY) THEN
            robotWS_State := SIM_JIG3PLACEDONE_WS;
        END_IF

    SIM_JIG3PLACEDONE_WS:
        IF WaitSync_Handler(E_WaitSync.OUTFEED_JIG3_PICKPLACE_DONE) THEN
            robotWS_State := PICK_DONE;
        END_IF

    PICK_DONE:
        ExecuteDetail_SIM := true;
        robotWS_State     := BOARD_READY_WS;
END_CASE
END_METHOD

METHOD ExecuteStep : BOOL
VAR_INPUT
    Step       : ST_CSV_Step;
    LineNumber : INT;
END_VAR
ExecuteStep := FALSE;

CASE Step.seqName OF
    E_CommandName.PickPlace:

        PickPlaceParse(Step, PickPlaceData);
        _PickPlaceDataToPass := PickPlaceData;
        // clear out array first
        Robot.Clear_DataToSend();

        // first entry is always step type
        Robot.RecipeData_ToSend[0] := E_CommandName.PickPlace;

        Robot.RecipeData_ToSend[1] := INT_TO_DINT(PickPlaceData.Number);

        Robot.RecipeData_ToSend[2] := REAL_TO_DINT(PickPlaceData.Length);

        Robot.RecipeData_ToSend[3] := REAL_TO_DINT(PickPlaceData.Width);

        Robot.RecipeData_ToSend[4] := REAL_TO_DINT(PickPlaceData.XPos);

        Robot.RecipeData_ToSend[5] := REAL_TO_DINT(PickPlaceData.YPos);

        Robot.RecipeData_ToSend[6] := REAL_TO_DINT(PickPlaceData.ZPos);

        Robot.RecipeData_ToSend[7] := REAL_TO_DINT(PickPlaceData.ZRot);

        Robot.RecipeData_ToSend[8] := INT_TO_DINT(PickPlaceData.ConvIndex);

        Robot.RecipeData_ToSend[9] := INT_TO_DINT(LineNumber);

        IF _InSimulation THEN
            IF ExecuteDetail_SIM(Step.seqID, LineNumber) THEN
                ExecuteStep := TRUE;
            END_IF
        ELSE
            IF ExecuteDetail(Step.seqID) THEN
                ExecuteStep := TRUE;
            END_IF
        END_IF

ELSE
    ExecuteStep := TRUE;

END_CASE
END_METHOD

METHOD HMIControl
VAR_INPUT
END_VAR
END_METHOD

//! @summary Basic module initialization logic
METHOD PROTECTED Initialize : BOOL;
VAR
    i                        : UDINT;
    varInfo                  : __SYSTEM.VAR_INFO;
    AllSubUnitsInitialized   : BOOL := TRUE;
    AllComponentsInitialized : BOOL := TRUE;
END_VAR

//! @description This method is called by <c>CyclicLogic()</c> as required
Initialize := FALSE;

CASE DescendantSequenceState OF
    0:
        RegisterComponent(Robot);

        _LogModeChanges         := FALSE;
        _LogStateChanges        := FALSE;
        DescendantSequenceState := DescendantSequenceState + 10;

    10:
        //Setup Custom modes here

        (*CustomModes(eMode                          :=,
                    sName                          :=,
                    bDisableClearing               :=,
                    bDisableStarting               :=,
                    bDisableSuspended              :=,
                    bDisableStopping               :=,
                    bDisableAborting               :=,
                    bDisableHolding                :=,
                    bDisableHeld                   :=,
                    bDisableUnholding              :=,
                    bDisableSuspending             :=,
                    bDisableUnsuspending           :=,
                    bDisableResetting              :=,
                    bDisableIdle                   :=,
                    bDisableCompleting             :=,
                    bDisableComplete               :=,
                    bEnableUnitModeChangeStopped   :=,
                    bEnableUnitModeChangeIdle      :=,
                    bEnableUnitModeChangeSuspended :=,
                    bEnableUnitModeChangeExecute   :=,
                    bEnableUnitModeChangeAborted   :=,
                    bEnableUnitModeChangeHeld      :=,
                    bEnableUnitModeChangeComplete  :=,
                    bError                         =>,
                    nErrorId                       =>);*)

        DescendantSequenceState := DescendantSequenceState + 10;

    20:
        //Copy Mode names

        FOR i := 1 TO 3 DO
            ModeNames[i] := F_UnitModeToString(UDINT_TO_DINT(i));
        END_FOR

        RegisterExternalController(Controller := fbControlSourceHMI);
        fbControlSourceHMI.CyclicLogic();
        DescendantSequenceState := DescendantSequenceState + 10;

    30:
        //Call the Super

        IF SUPER^.Initialize() THEN
            DescendantSequenceState := DescendantSequenceState + 10;
        END_IF

    40:
        Initialize := TRUE;
END_CASE
END_METHOD

METHOD UI_MessageBox : BOOL
VAR_INPUT
END_VAR

VAR
    result : USINT;
END_VAR
IF Robot.Handshake.IN.ErrorPresent THEN
    CASE Robot.Handshake.IN.MessageNumber OF

        //////////////////////////// ASSEMBLY PLC ERRORS ////////////////////////////
        0:

            // Idle State Should not have an error of 0

            ////////// 1-29 PROCESS ERRORS /////////

            // Note: The code for messages 1 and 2 is commented out, so we skip them.

        3:
            // PrePlate ERROR_PROCESSING_DATA
            result := RaiseMessageBox(Header   := 'Processing Data Error ASSEMBLY',
                                      Message1 := 'PLC Received same file twice from SAM',
                                      Message2 := 'Choose RETRY to retry data processing',
                                      Message3 := 'Choose CONTINUE to proceed anyways',
                                      Btn3     := 'RETRY',
                                      Btn5     := 'CONTINUE',
                                      Severity := TcEventSeverity.Error);

        15:
            // Press Error Detected
            result := RaiseMessageBox(Header   := 'Press Error Detected',
                                      Message1 := 'Select CLEAR to clear error and send press back to idle',
                                      Btn3     := 'CLEAR',
                                      Severity := TcEventSeverity.Error);

        16:
            // Waiting on Press
            result := RaiseMessageBox(Header   := 'Waiting on Press',
                                      Message1 := 'Waiting for press to be fully retracted and in IDLE state',
                                      Message3 := 'Select RESET to cycle/retract press',
                                      Btn3     := 'RESET',
                                      Severity := TcEventSeverity.Error);

        19:
            // test alarm
            result := RaiseMessageBox(Header   := 'test alarm',
                                      Message1 := 'Message1',
                                      Message2 := 'Message2',
                                      Message3 := 'Message3',
                                      Message4 := 'Message4',
                                      Message5 := 'Message5',
                                      Btn1     := 'button 1',
                                      Btn2     := 'button 2',
                                      Btn3     := 'button 3',
                                      Btn4     := 'button 4',
                                      Btn5     := 'button 5',
                                      Severity := TcEventSeverity.Error);

        26:
            // System Suspended
            result := RaiseMessageBox(Header   := 'System Suspended',
                                      Message1 := 'Press OK to clear message',
                                      Message3 := 'Clear any active errors on carriages or robots and press Resume to continue',
                                      Btn3     := 'OK',
                                      Severity := TcEventSeverity.Error);

            ////////// 30-59 ROBOT ERRORS /////////
        30:
            // Outfeed Robot Stopped
            result := RaiseMessageBox(Header   := 'Outfeed Robot Stopped',
                                      Message1 := 'Outfeed robot crashed/stopped',
                                      Message2 := 'Check assembly robot area to make sure nothing is obstructing the robot',
                                      Message3 := 'Select OK to dismiss error message',
                                      Btn3     := 'OK',
                                      Severity := TcEventSeverity.Error);

        31:
            // Outfeed Robot Error
            result := RaiseMessageBox(Header   := 'Outfeed Robot Error',
                                      Message1 := 'Check robots teach pendant to see what the issue is.',
                                      Message2 := 'Select CONTINUE when the robot is ready to retry.',
                                      Btn5     := 'CONTINUE',
                                      Severity := TcEventSeverity.Error);

        35:
            // Light Curtain Tripped
            result := RaiseMessageBox(Header   := 'Light Curtain Tripped',
                                      Message1 := 'Outfeed light curtains detected movement',
                                      Message2 := 'Make sure outfeed area is clear before resuming',
                                      Message3 := 'Select OK to dismiss error message',
                                      Btn3     := 'OK',
                                      Severity := TcEventSeverity.Error);

        38:
            // EOAT Failed to Pick Board
            result := RaiseMessageBox(Header   := 'EOAT Failed to Pick Board',
                                      Message1 := 'Choose RETRY to repick board',
                                      Message3 := 'Choose OVERRIDE to continue with pick',
                                      Btn3     := 'RETRY',
                                      Btn4     := 'OVERRIDE',
                                      Severity := TcEventSeverity.Error);

        48:
            // Check board height
            result := RaiseMessageBox(Header   := 'Check board height',
                                      Message1 := '',
                                      Message2 := 'Pick motor not at correct height',
                                      Message3 := 'Check to make sure correct board was loaded and teeth are embedded in the wood',
                                      Message5 := 'If correct board is loaded then press OVERRIDE to continue',
                                      Btn1     := 'OVERRIDE',
                                      Severity := TcEventSeverity.Error);

        51:
            // confirm material has been cleared
            result := RaiseMessageBox(Header   := 'Remove Material from Assembly Conveyors',
                                      Message1 := 'Remove any boards from the Assembly area',
                                      Message2 := 'Select OK when system is ready to continue',
                                      Btn5     := 'OK',
                                      Severity := TcEventSeverity.Error);

        53:
            // Skip Press?
            result := RaiseMessageBox(Header   := 'Skip Press?',
                                      Message1 := 'SKIP wills skip all press motion and use a 2.5s timer to simulate press',
                                      Message3 := 'PRESS will press like normal',
                                      Btn3     := 'SKIP',
                                      Btn5     := 'PRESS',
                                      Severity := TcEventSeverity.Error);

        54:
            // Velocity
            result := RaiseMessageBox(Header   := 'Velocity',
                                      Message1 := 'This is the speed the carriages will run',
                                      Btn2     := '2000',
                                      Btn3     := '3000',
                                      Btn4     := '4000',
                                      Severity := TcEventSeverity.Error);

        55:
            // Are You Sure?
            result := RaiseMessageBox(Header   := 'Are You Sure?',
                                      Message1 := '4000 is pretty quick speed racer',
                                      Btn2     := 'YES',
                                      Btn3     := 'NO',
                                      Btn4     := 'MAYBE',
                                      Severity := TcEventSeverity.Error);

        56:
            // No System Config File Loaded
            result := RaiseMessageBox(Header   := 'No System Config File Loaded',
                                      Message1 := 'Load in sys config file and retry',
                                      Btn5     := 'RETRY',
                                      Severity := TcEventSeverity.Error);

        70:
            // Assembly Abort Requested
            result := RaiseMessageBox(Header   := 'Assembly Abort Requested',
                                      Message1 := CONCAT('How do you want to abort truss ', ''),
                                      Message2 := 'Abort will scrap the truss',
                                      Message3 := 'Manual will stop running the truss but allow you to manually build it.',
                                      Message4 := 'Retry will stop running the truss and requeue it in SAM',
                                      Btn2     := 'ABORT',
                                      Btn3     := 'MANUAL',
                                      Btn4     := 'RETRY',
                                      Severity := TcEventSeverity.Error);

        71:
            // Eject 1 Abort Requested
            result := RaiseMessageBox(Header   := 'Eject 1 Abort Requested',
                                      Message1 := CONCAT('How do you want to abort truss ', ''),
                                      Message2 := 'Abort will scrap the truss',
                                      Message3 := 'Manual will stop running the truss but allow you to manually build it.',
                                      Message4 := 'Retry will stop running the truss and requeue it in SAM',
                                      Message5 := 'Select CANCEL to continue build',
                                      Btn2     := 'ABORT',
                                      Btn3     := 'MANUAL',
                                      Btn4     := 'RETRY',
                                      Btn5     := 'CANCEL',
                                      Severity := TcEventSeverity.Error);

        72:
            // Eject 2 Abort Requested
            result := RaiseMessageBox(Header   := 'Eject 2 Abort Requested',
                                      Message1 := CONCAT('How do you want to abort truss ', ''),
                                      Message2 := 'Abort will scrap the truss',
                                      Message3 := 'Manual will stop running the truss but allow you to manually build it.',
                                      Message4 := 'Retry will stop running the truss and requeue it in SAM',
                                      Btn2     := 'ABORT',
                                      Btn3     := 'MANUAL',
                                      Btn4     := 'RETRY',
                                      Severity := TcEventSeverity.Error);

        73:
            // Assembly AirPressure
            result := RaiseMessageBox(Header   := 'Low Air Pressure At Outfeed',
                                      Message1 := 'Pressure near Assembly is low',
                                      Message3 := 'Check dump valve and sensor',
                                      Message5 := 'Press OK to test again',
                                      Btn1     := 'OK',
                                      Severity := TcEventSeverity.Error);

        90:
            // Board Not detected
            result := RaiseMessageBox(Header   := 'No Board Detected.',
                                      Message1 := 'Choose RETRY to repick board',
                                      Message3 := 'Choose OVERRIDE to continue with pick',
                                      Btn3     := 'RETRY',
                                      Btn4     := 'Override',
                                      Severity := TcEventSeverity.Error);
        92:
            // Board Not detected
            result := RaiseMessageBox(Header   := 'Check Board.',
                                      Message1 := 'Choose Continue to retry picking board',
                                      Btn3     := 'CONTINUE',
                                      Severity := TcEventSeverity.Error);

        93:
            // Board Not detected
            result := RaiseMessageBox(Header   := 'Board Not Detected When Placing',
                                      Message1 := 'Verify board is being held',
                                      Message2 := 'If there is no board make sure board is placed fully on conveyor',
                                      Message3 := 'If there is no board, check if robot track is clear',
                                      Message4 := 'Press OK to continue',
                                      Btn5     := 'OK',
                                      Severity := TcEventSeverity.Error);

    ELSE
        // Not Valid Message Number

        // The original code appends the ErrorNumber integer to the message.

        // We'll keep the same logic, but we can store it as a separate or inline string.

        // For demonstration, we directly pass in the integer, though we normally would do

        // a conversion. We'll just label it as an unknown message.
        result := RaiseMessageBox(Header   := 'Not Valid Message Number',
                                  Message1 := CONCAT('UIMessageBox was sent message number: ', UINT_TO_STRING(Robot.Handshake.IN.MessageNumber)),
                                  Message3 := 'Contact Support to update message number.',
                                  Btn1     := 'EXIT MSG',
                                  Severity := TcEventSeverity.Error);
    END_CASE;

    IF result <> 0 THEN
        Robot.Handshake.OUT.MessageSolution    := result;
        Robot.Handshake.OUT.MessageAcknowledge := TRUE;
    END_IF
ELSE
    Robot.Handshake.OUT.MessageSolution    := 0;
    Robot.Handshake.OUT.MessageAcknowledge := FALSE;
END_IF;
END_METHOD

